// TIA Portal V17 export
// export: Created 2024-06-14T09:52:58.9808405Z, ExportSetting WithDefaults, DisplayName Totally Integrated Automation Portal, DisplayVersion V17, DisplayName TIA Portal Openness, DisplayVersion V17, DisplayName TIA Portal Version Control Interface, DisplayVersion V17, DisplayName Simotion SCOUT TIA, DisplayVersion 5.4.3.0, DisplayName SINAMICS Startdrive Advanced, DisplayVersion V17 SP1 Update 1, DisplayName SINAMICS Startdrive G110M, G120, G120C, G120D, G120P, G115D, DisplayVersion V17 SP1 Update 1, DisplayName SINAMICS Startdrive G130, G150, S120, S150, SINAMICS MV, S210, DisplayVersion V17 SP1 Update 1, DisplayName STEP 7 Professional, DisplayVersion V17, DisplayName STEP 7 Safety, DisplayVersion V17, DisplayName WinCC Professional, DisplayVersion V17
FUNCTION "STATION S1" : Void   // FC3, LAD
{ S7_Optimized_Access := 'TRUE' }
VERSION : 0.1
// stored: AutoNumber true, IsIECCheckEnabled false, SetENOAutomatically false, UDAEnableTagReadback false
   VAR_INPUT
      CYLINDER_POS_IN : Bool;
      INxcommercial_Cy : Bool;
      "CYLINDER EXIT" : Bool;
      sensor_line_1 : Bool;
      sensor_line_2 : Bool;
   END_VAR
   VAR_OUTPUT
      OUTxCylinder_Count : Bool;
      STOPPRER : Bool;
      Tare_Weight_Error : Bool;
      Enter_Tare_weight : Bool;
      Cylinder_type_error : Bool;
      data_count : Int;
   END_VAR
   VAR_IN_OUT
      S9_Array_copy : Int;
   END_VAR
   VAR_TEMP
      TRUCK : String;
      Start : Bool;
      copied_item : Int;
      Ret_val_1 : Int;
      Out_RD : DTL;
      Difference_Domestic_Cy : Real;
      Difference_commercial_Cy : Real;
      set_bit : Bool;
      Full_Wieght_Difference : Real;
      idx1 : Int;
      idx2 : Int;
      idx3 : Int;
      idx4 : Int;
      idx5 : Int;
      idx6 : Int;
      idx7 : Int;
      Gross_Weight : Real;
      "cylinder ok" : Bool;
      ptrig : Bool;
      ptrig_1 : Bool;
      ptrig_2 : Bool;
      TEMP : Int;
      pass : Bool;
      FILL_DB : Bool;
      TEMP_1 : Int;
      TEMP_2 : Int;
      TEMP_3 : Int;
      TEMP_4 : Int;
      TEMP_5 : Int;
      TEMP_6 : Int;
      TEMP_7 : Int;
      TEMP_8 : Int;
      TEMP_9 : Int;
      TEMP_10 : Int;
      TEMP_11 : Int;
      TEMP_12 : Int;
      TEMP_13 : Int;
      TEMP_14 : Int;
   END_VAR
   VAR_TEMP   // added for the SCL form of the ladder/FBD networks
      _w1 : Bool;
      _w2 : Bool;
      _w3 : Bool;
      _w4 : Bool;
      _w5 : Bool;
      _w6 : Bool;
      _w7 : Bool;
      _w8 : Bool;
      _w9 : Bool;
   END_VAR
BEGIN

REGION Network 1: Cylinder_Count
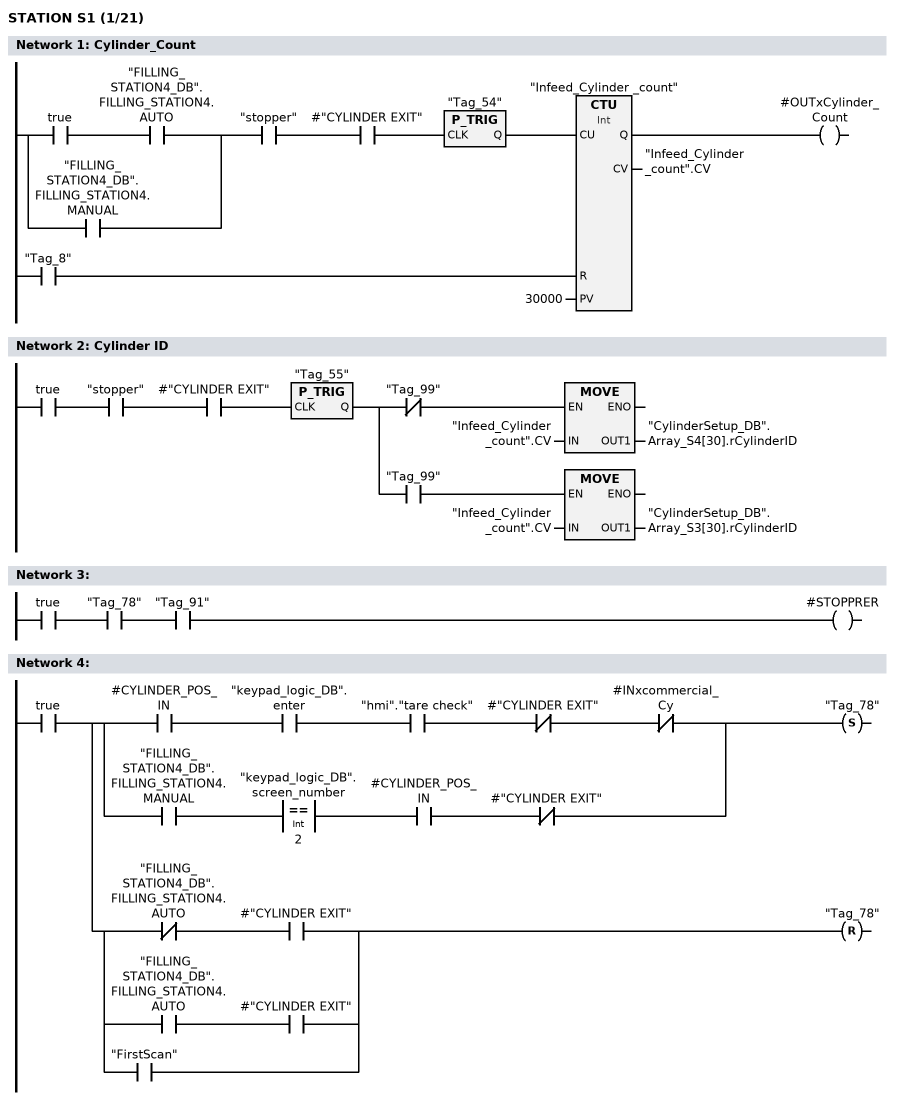
   RUNG wire#powerrail
      Contact( true )
      Contact( "FILLING_STATION4_DB".FILLING_STATION4.AUTO )
      wire#w1
      Contact( "stopper" )
      Contact( #"CYLINDER EXIT" )
      P_Trig( "Tag_54" )
      { S7_Templates := "value_type := Int" } "Infeed_Cylinder _count".CTU(r := wire#w2, pv := 30000, cv => "Infeed_Cylinder _count".CV)
      Coil( #OUTxCylinder_Count )
   END_RUNG
   RUNG wire#powerrail
      Contact( "FILLING_STATION4_DB".FILLING_STATION4.MANUAL )
   END_RUNG wire#w1
   RUNG wire#powerrail
      Contact( "Tag_8" )
   END_RUNG wire#w2
   // the same network as SCL:
   #_w1 := ((true AND "FILLING_STATION4_DB".FILLING_STATION4.AUTO) OR "FILLING_STATION4_DB".FILLING_STATION4.MANUAL) AND "stopper" AND #"CYLINDER EXIT";
   #_w2 := #_w1 AND NOT "Tag_54";   // rising edge
   "Tag_54" := #_w1;
   "Infeed_Cylinder _count".CTU(CU := #_w2, R := "Tag_8", PV := 30000, CV => "Infeed_Cylinder _count".CV);
   #OUTxCylinder_Count := "Infeed_Cylinder _count".Q;
END_REGION

REGION Network 2: Cylinder ID
   RUNG wire#powerrail
      Contact( true )
      Contact( "stopper" )
      Contact( #"CYLINDER EXIT" )
      P_Trig( "Tag_55" )
      wire#w1
      I_Contact( "Tag_99" )
      Move(in := "Infeed_Cylinder _count".CV, out1 => "CylinderSetup_DB".Array_S4[30].rCylinderID)
   END_RUNG
   RUNG wire#w1
      Contact( "Tag_99" )
      Move(in := "Infeed_Cylinder _count".CV, out1 => "CylinderSetup_DB".Array_S3[30].rCylinderID)
   END_RUNG
   // the same network as SCL:
   #_w1 := true AND "stopper" AND #"CYLINDER EXIT";
   #_w2 := #_w1 AND NOT "Tag_55";   // rising edge
   "Tag_55" := #_w1;
   IF #_w2 AND NOT "Tag_99" THEN
       "CylinderSetup_DB".Array_S4[30].rCylinderID := "Infeed_Cylinder _count".CV;
   END_IF;
   IF #_w2 AND "Tag_99" THEN
       "CylinderSetup_DB".Array_S3[30].rCylinderID := "Infeed_Cylinder _count".CV;
   END_IF;
END_REGION

REGION Network 3
   RUNG wire#powerrail
      Contact( true )
      Contact( "Tag_78" )
      Contact( "Tag_91" )
      Coil( #STOPPRER )
   END_RUNG
   // the same network as SCL:
   #STOPPRER := true AND "Tag_78" AND "Tag_91";
END_REGION

REGION Network 4
   RUNG wire#powerrail
      Contact( true )
      wire#w1
      Contact( #CYLINDER_POS_IN )
      Contact( "keypad_logic_DB".enter )
      Contact( "hmi"."tare check" )
      I_Contact( #"CYLINDER EXIT" )
      I_Contact( #INxcommercial_Cy )
      wire#w2
      S_Coil( "Tag_78" )
   END_RUNG
   RUNG wire#w1
      Contact( "FILLING_STATION4_DB".FILLING_STATION4.MANUAL )
      { S7_Templates := "SrcType := Int" } EQ_Contact(in1 := "keypad_logic_DB".screen_number, in2 := 2)
      Contact( #CYLINDER_POS_IN )
      I_Contact( #"CYLINDER EXIT" )
   END_RUNG wire#w2
   RUNG wire#w1
      I_Contact( "FILLING_STATION4_DB".FILLING_STATION4.AUTO )
      Contact( #"CYLINDER EXIT" )
      wire#w3
      R_Coil( "Tag_78" )
   END_RUNG
   RUNG wire#w1
      Contact( "FILLING_STATION4_DB".FILLING_STATION4.AUTO )
      Contact( #"CYLINDER EXIT" )
   END_RUNG wire#w3
   RUNG wire#w1
      Contact( "FirstScan" )
   END_RUNG wire#w3
   // the same network as SCL:
   IF true AND ((#CYLINDER_POS_IN AND "keypad_logic_DB".enter AND "hmi"."tare check" AND NOT #"CYLINDER EXIT" AND NOT #INxcommercial_Cy) OR ("FILLING_STATION4_DB".FILLING_STATION4.MANUAL AND ("keypad_logic_DB".screen_number = 2) AND #CYLINDER_POS_IN AND NOT #"CYLINDER EXIT")) THEN
       "Tag_78" := TRUE;
   END_IF;
   IF true AND ((NOT "FILLING_STATION4_DB".FILLING_STATION4.AUTO AND #"CYLINDER EXIT") OR ("FILLING_STATION4_DB".FILLING_STATION4.AUTO AND #"CYLINDER EXIT") OR "FirstScan") THEN
       "Tag_78" := FALSE;
   END_IF;
END_REGION

REGION Network 5: Domestic_Cylinder_Details
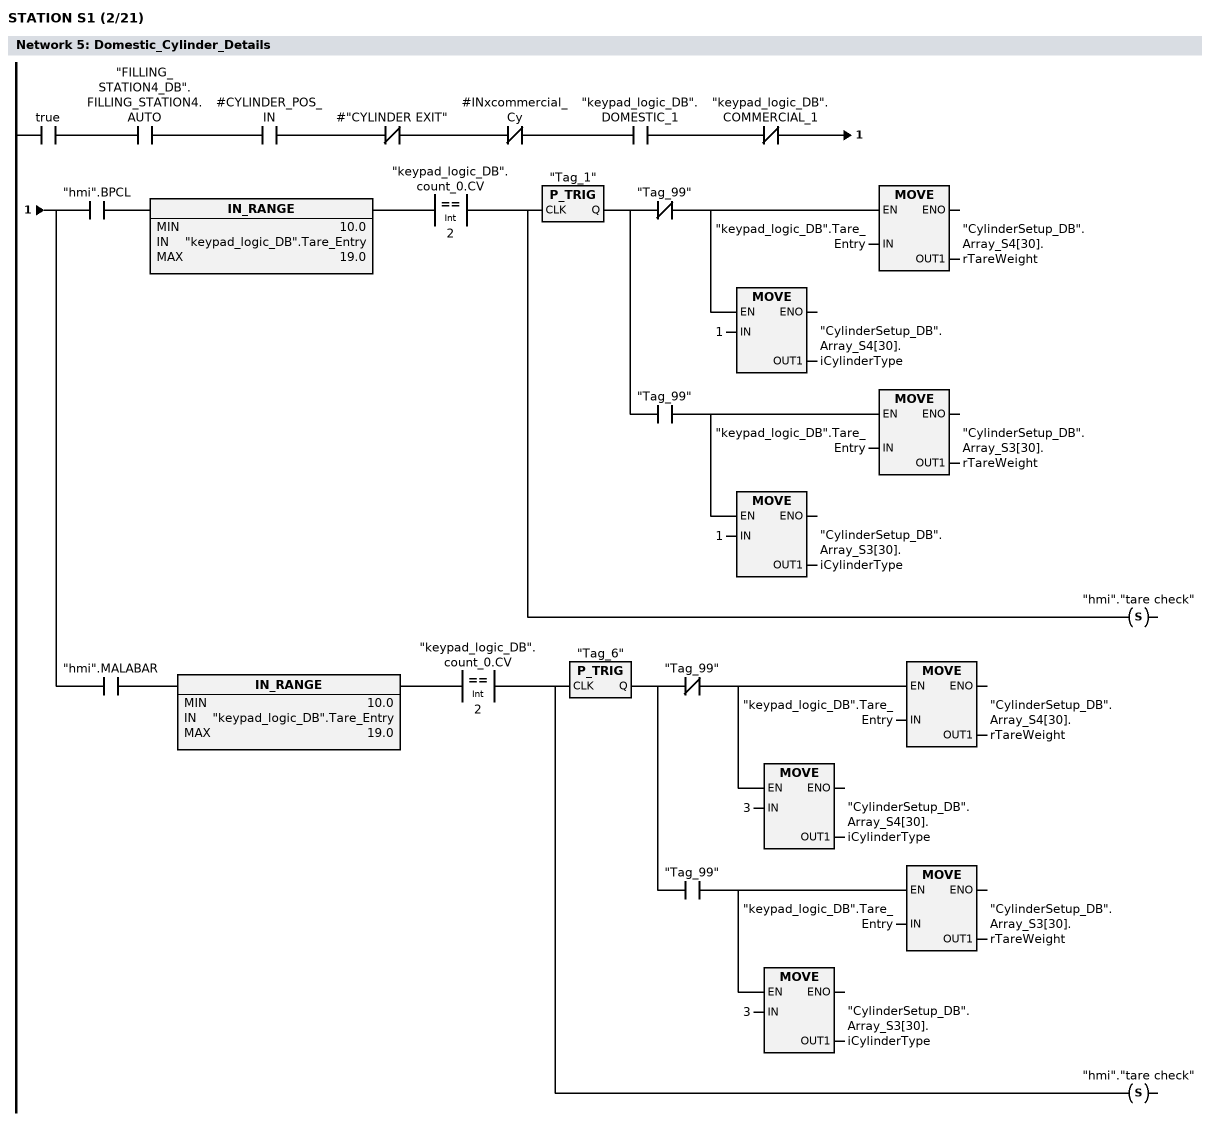
   RUNG wire#powerrail
      Contact( true )
      Contact( "FILLING_STATION4_DB".FILLING_STATION4.AUTO )
      Contact( #CYLINDER_POS_IN )
      I_Contact( #"CYLINDER EXIT" )
      I_Contact( #INxcommercial_Cy )
      Contact( "keypad_logic_DB".DOMESTIC_1 )
      I_Contact( "keypad_logic_DB".COMMERCIAL_1 )
      wire#w1
      Contact( "hmi".BPCL )
      { S7_Templates := "SrcType := Real" } InRange(min := 10.0, in := "keypad_logic_DB".Tare_Entry, max := 19.0)
      { S7_Templates := "SrcType := Int" } EQ_Contact(in1 := "keypad_logic_DB".count_0.CV, in2 := 2)
      wire#w2
      P_Trig( "Tag_1" )
      wire#w3
      I_Contact( "Tag_99" )
      wire#w4
      Move(in := "keypad_logic_DB".Tare_Entry, out1 => "CylinderSetup_DB".Array_S4[30].rTareWeight)
   END_RUNG
   RUNG wire#w4
      Move(in := 1, out1 => "CylinderSetup_DB".Array_S4[30].iCylinderType)
   END_RUNG
   RUNG wire#w3
      Contact( "Tag_99" )
      wire#w5
      Move(in := "keypad_logic_DB".Tare_Entry, out1 => "CylinderSetup_DB".Array_S3[30].rTareWeight)
   END_RUNG
   RUNG wire#w5
      Move(in := 1, out1 => "CylinderSetup_DB".Array_S3[30].iCylinderType)
   END_RUNG
   RUNG wire#w2
      S_Coil( "hmi"."tare check" )
   END_RUNG
   RUNG wire#w1
      Contact( "hmi".MALABAR )
      { S7_Templates := "SrcType := Real" } InRange(min := 10.0, in := "keypad_logic_DB".Tare_Entry, max := 19.0)
      { S7_Templates := "SrcType := Int" } EQ_Contact(in1 := "keypad_logic_DB".count_0.CV, in2 := 2)
      wire#w6
      P_Trig( "Tag_6" )
      wire#w7
      I_Contact( "Tag_99" )
      wire#w8
      Move(in := "keypad_logic_DB".Tare_Entry, out1 => "CylinderSetup_DB".Array_S4[30].rTareWeight)
   END_RUNG
   RUNG wire#w8
      Move(in := 3, out1 => "CylinderSetup_DB".Array_S4[30].iCylinderType)
   END_RUNG
   RUNG wire#w7
      Contact( "Tag_99" )
      wire#w9
      Move(in := "keypad_logic_DB".Tare_Entry, out1 => "CylinderSetup_DB".Array_S3[30].rTareWeight)
   END_RUNG
   RUNG wire#w9
      Move(in := 3, out1 => "CylinderSetup_DB".Array_S3[30].iCylinderType)
   END_RUNG
   RUNG wire#w6
      S_Coil( "hmi"."tare check" )
   END_RUNG
   // the same network as SCL:
   #_w1 := true AND "FILLING_STATION4_DB".FILLING_STATION4.AUTO AND #CYLINDER_POS_IN AND NOT #"CYLINDER EXIT" AND NOT #INxcommercial_Cy AND "keypad_logic_DB".DOMESTIC_1 AND NOT "keypad_logic_DB".COMMERCIAL_1;
   #_w2 := #_w1 AND "hmi".BPCL AND (10.0 <= "keypad_logic_DB".Tare_Entry) AND ("keypad_logic_DB".Tare_Entry <= 19.0) AND ("keypad_logic_DB".count_0.CV = 2);
   #_w3 := #_w2 AND NOT "Tag_1";   // rising edge
   "Tag_1" := #_w2;
   IF #_w3 AND NOT "Tag_99" THEN
       "CylinderSetup_DB".Array_S4[30].rTareWeight := "keypad_logic_DB".Tare_Entry;
       "CylinderSetup_DB".Array_S4[30].iCylinderType := 1;
   END_IF;
   IF #_w3 AND "Tag_99" THEN
       "CylinderSetup_DB".Array_S3[30].rTareWeight := "keypad_logic_DB".Tare_Entry;
       "CylinderSetup_DB".Array_S3[30].iCylinderType := 1;
   END_IF;
   IF #_w2 THEN "hmi"."tare check" := TRUE; END_IF;
   #_w4 := #_w1 AND "hmi".MALABAR AND (10.0 <= "keypad_logic_DB".Tare_Entry) AND ("keypad_logic_DB".Tare_Entry <= 19.0) AND ("keypad_logic_DB".count_0.CV = 2);
   #_w5 := #_w4 AND NOT "Tag_6";   // rising edge
   "Tag_6" := #_w4;
   IF #_w5 AND NOT "Tag_99" THEN
       "CylinderSetup_DB".Array_S4[30].rTareWeight := "keypad_logic_DB".Tare_Entry;
       "CylinderSetup_DB".Array_S4[30].iCylinderType := 3;
   END_IF;
   IF #_w5 AND "Tag_99" THEN
       "CylinderSetup_DB".Array_S3[30].rTareWeight := "keypad_logic_DB".Tare_Entry;
       "CylinderSetup_DB".Array_S3[30].iCylinderType := 3;
   END_IF;
   IF #_w4 THEN "hmi"."tare check" := TRUE; END_IF;
END_REGION

REGION Network 6: DOMESTIC_ALARM
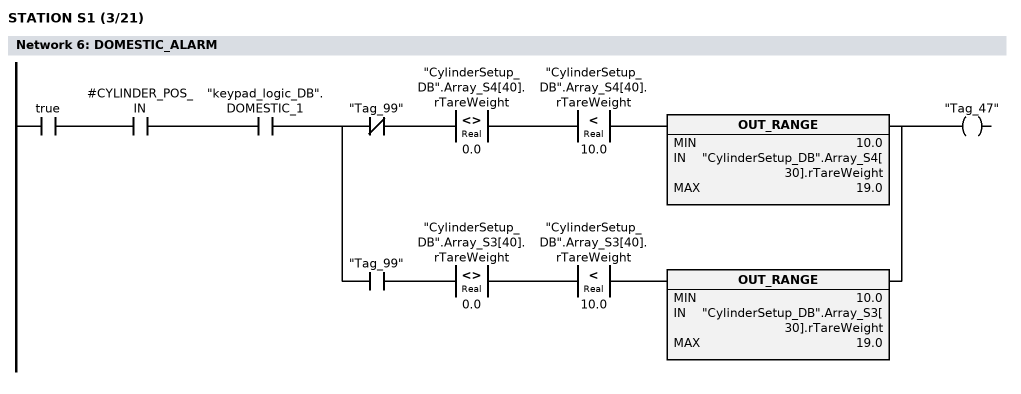
   "Tag_47" := true AND #CYLINDER_POS_IN AND "keypad_logic_DB".DOMESTIC_1 AND ((NOT "Tag_99" AND ("CylinderSetup_DB".Array_S4[40].rTareWeight <> 0.0) AND ("CylinderSetup_DB".Array_S4[40].rTareWeight < 10.0) AND (("CylinderSetup_DB".Array_S4[30].rTareWeight < 10.0) OR ("CylinderSetup_DB".Array_S4[30].rTareWeight > 19.0))) OR ("Tag_99" AND ("CylinderSetup_DB".Array_S3[40].rTareWeight <> 0.0) AND ("CylinderSetup_DB".Array_S3[40].rTareWeight < 10.0) AND (("CylinderSetup_DB".Array_S3[30].rTareWeight < 10.0) OR ("CylinderSetup_DB".Array_S3[30].rTareWeight > 19.0))));
END_REGION

REGION Network 7: Commercial_Cylinder_Details
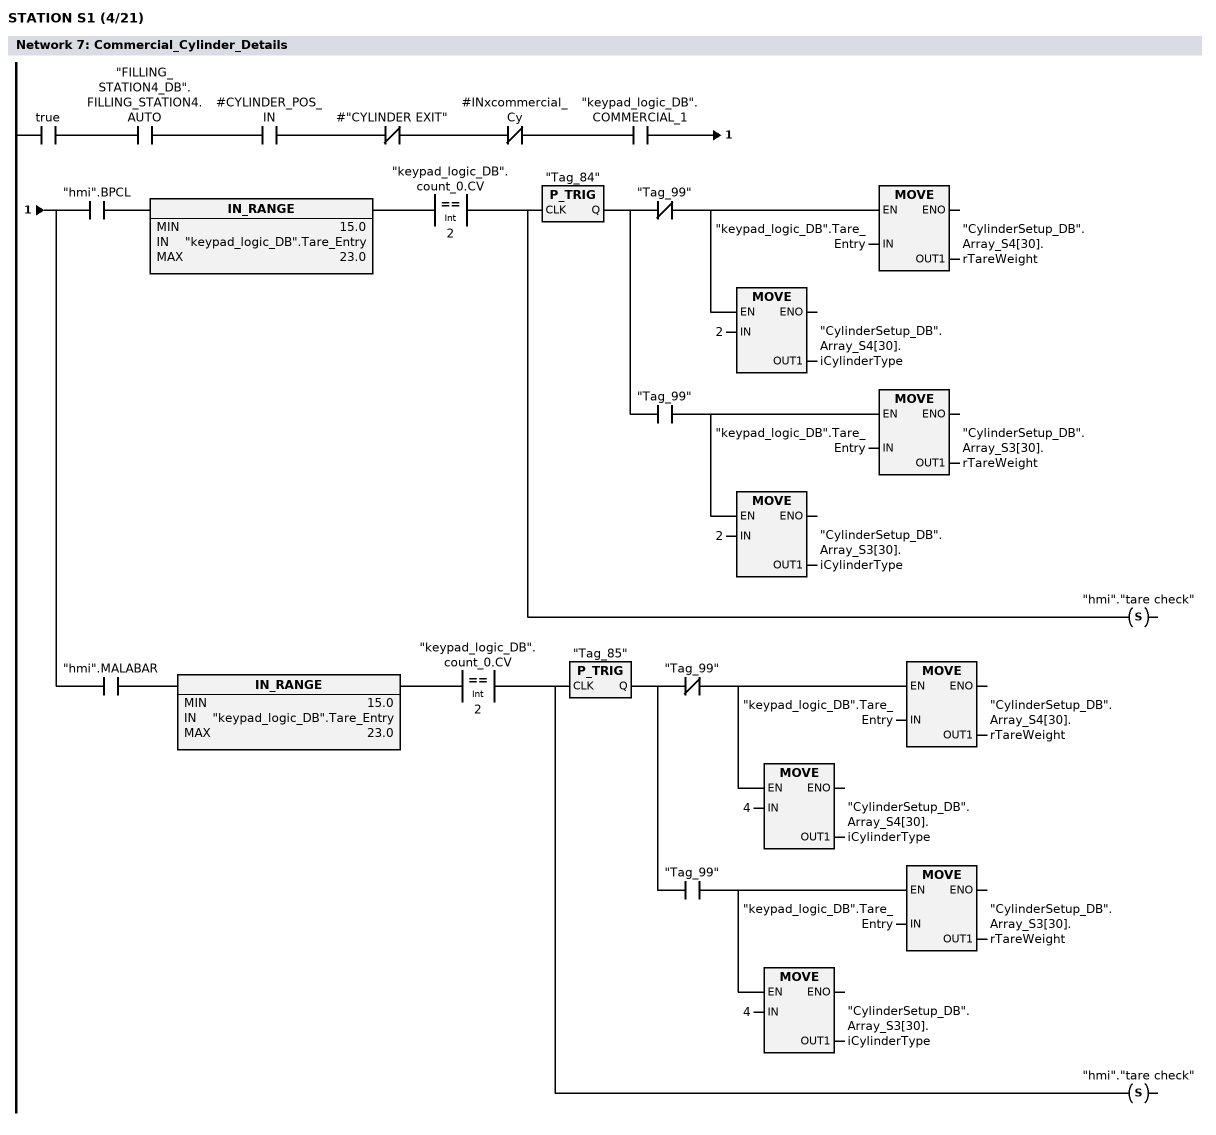
   RUNG wire#powerrail
      Contact( true )
      Contact( "FILLING_STATION4_DB".FILLING_STATION4.AUTO )
      Contact( #CYLINDER_POS_IN )
      I_Contact( #"CYLINDER EXIT" )
      I_Contact( #INxcommercial_Cy )
      Contact( "keypad_logic_DB".COMMERCIAL_1 )
      wire#w1
      Contact( "hmi".BPCL )
      { S7_Templates := "SrcType := Real" } InRange(min := 15.0, in := "keypad_logic_DB".Tare_Entry, max := 23.0)
      { S7_Templates := "SrcType := Int" } EQ_Contact(in1 := "keypad_logic_DB".count_0.CV, in2 := 2)
      wire#w2
      P_Trig( "Tag_84" )
      wire#w3
      I_Contact( "Tag_99" )
      wire#w4
      Move(in := "keypad_logic_DB".Tare_Entry, out1 => "CylinderSetup_DB".Array_S4[30].rTareWeight)
   END_RUNG
   RUNG wire#w4
      Move(in := 2, out1 => "CylinderSetup_DB".Array_S4[30].iCylinderType)
   END_RUNG
   RUNG wire#w3
      Contact( "Tag_99" )
      wire#w5
      Move(in := "keypad_logic_DB".Tare_Entry, out1 => "CylinderSetup_DB".Array_S3[30].rTareWeight)
   END_RUNG
   RUNG wire#w5
      Move(in := 2, out1 => "CylinderSetup_DB".Array_S3[30].iCylinderType)
   END_RUNG
   RUNG wire#w2
      S_Coil( "hmi"."tare check" )
   END_RUNG
   RUNG wire#w1
      Contact( "hmi".MALABAR )
      { S7_Templates := "SrcType := Real" } InRange(min := 15.0, in := "keypad_logic_DB".Tare_Entry, max := 23.0)
      { S7_Templates := "SrcType := Int" } EQ_Contact(in1 := "keypad_logic_DB".count_0.CV, in2 := 2)
      wire#w6
      P_Trig( "Tag_85" )
      wire#w7
      I_Contact( "Tag_99" )
      wire#w8
      Move(in := "keypad_logic_DB".Tare_Entry, out1 => "CylinderSetup_DB".Array_S4[30].rTareWeight)
   END_RUNG
   RUNG wire#w8
      Move(in := 4, out1 => "CylinderSetup_DB".Array_S4[30].iCylinderType)
   END_RUNG
   RUNG wire#w7
      Contact( "Tag_99" )
      wire#w9
      Move(in := "keypad_logic_DB".Tare_Entry, out1 => "CylinderSetup_DB".Array_S3[30].rTareWeight)
   END_RUNG
   RUNG wire#w9
      Move(in := 4, out1 => "CylinderSetup_DB".Array_S3[30].iCylinderType)
   END_RUNG
   RUNG wire#w6
      S_Coil( "hmi"."tare check" )
   END_RUNG
   // the same network as SCL:
   #_w1 := true AND "FILLING_STATION4_DB".FILLING_STATION4.AUTO AND #CYLINDER_POS_IN AND NOT #"CYLINDER EXIT" AND NOT #INxcommercial_Cy AND "keypad_logic_DB".COMMERCIAL_1;
   #_w2 := #_w1 AND "hmi".BPCL AND (15.0 <= "keypad_logic_DB".Tare_Entry) AND ("keypad_logic_DB".Tare_Entry <= 23.0) AND ("keypad_logic_DB".count_0.CV = 2);
   #_w3 := #_w2 AND NOT "Tag_84";   // rising edge
   "Tag_84" := #_w2;
   IF #_w3 AND NOT "Tag_99" THEN
       "CylinderSetup_DB".Array_S4[30].rTareWeight := "keypad_logic_DB".Tare_Entry;
       "CylinderSetup_DB".Array_S4[30].iCylinderType := 2;
   END_IF;
   IF #_w3 AND "Tag_99" THEN
       "CylinderSetup_DB".Array_S3[30].rTareWeight := "keypad_logic_DB".Tare_Entry;
       "CylinderSetup_DB".Array_S3[30].iCylinderType := 2;
   END_IF;
   IF #_w2 THEN "hmi"."tare check" := TRUE; END_IF;
   #_w4 := #_w1 AND "hmi".MALABAR AND (15.0 <= "keypad_logic_DB".Tare_Entry) AND ("keypad_logic_DB".Tare_Entry <= 23.0) AND ("keypad_logic_DB".count_0.CV = 2);
   #_w5 := #_w4 AND NOT "Tag_85";   // rising edge
   "Tag_85" := #_w4;
   IF #_w5 AND NOT "Tag_99" THEN
       "CylinderSetup_DB".Array_S4[30].rTareWeight := "keypad_logic_DB".Tare_Entry;
       "CylinderSetup_DB".Array_S4[30].iCylinderType := 4;
   END_IF;
   IF #_w5 AND "Tag_99" THEN
       "CylinderSetup_DB".Array_S3[30].rTareWeight := "keypad_logic_DB".Tare_Entry;
       "CylinderSetup_DB".Array_S3[30].iCylinderType := 4;
   END_IF;
   IF #_w4 THEN "hmi"."tare check" := TRUE; END_IF;
END_REGION

REGION Network 8: COMMERCIAL_ALARM
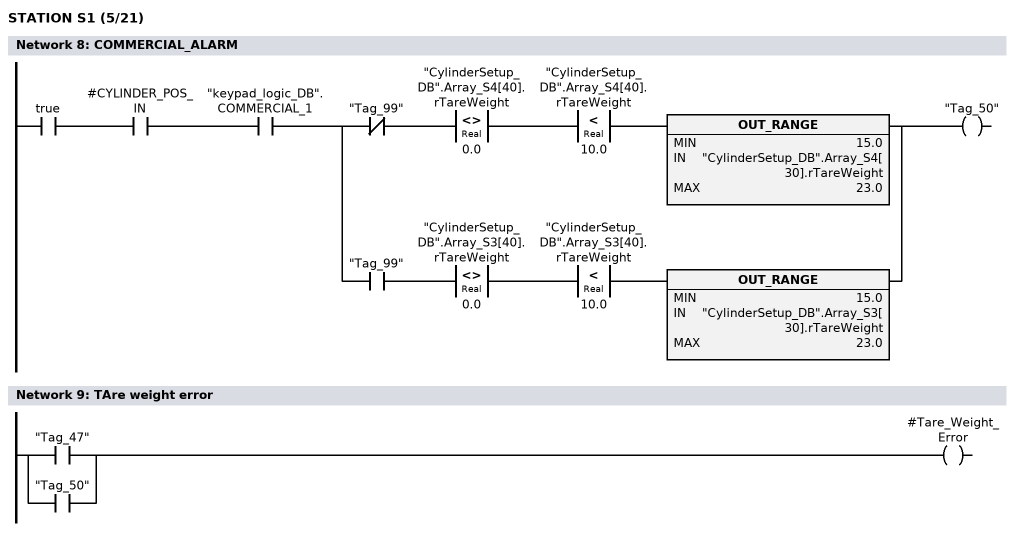
   "Tag_50" := true AND #CYLINDER_POS_IN AND "keypad_logic_DB".COMMERCIAL_1 AND ((NOT "Tag_99" AND ("CylinderSetup_DB".Array_S4[40].rTareWeight <> 0.0) AND ("CylinderSetup_DB".Array_S4[40].rTareWeight < 10.0) AND (("CylinderSetup_DB".Array_S4[30].rTareWeight < 15.0) OR ("CylinderSetup_DB".Array_S4[30].rTareWeight > 23.0))) OR ("Tag_99" AND ("CylinderSetup_DB".Array_S3[40].rTareWeight <> 0.0) AND ("CylinderSetup_DB".Array_S3[40].rTareWeight < 10.0) AND (("CylinderSetup_DB".Array_S3[30].rTareWeight < 15.0) OR ("CylinderSetup_DB".Array_S3[30].rTareWeight > 23.0))));
END_REGION

REGION Network 9: TAre weight error
   RUNG wire#powerrail
      Contact( "Tag_47" )
      wire#w1
      Coil( #Tare_Weight_Error )
   END_RUNG
   RUNG wire#powerrail
      Contact( "Tag_50" )
   END_RUNG wire#w1
   // the same network as SCL:
   #Tare_Weight_Error := "Tag_47" OR "Tag_50";
END_REGION

REGION Network 10: S4_Array Move
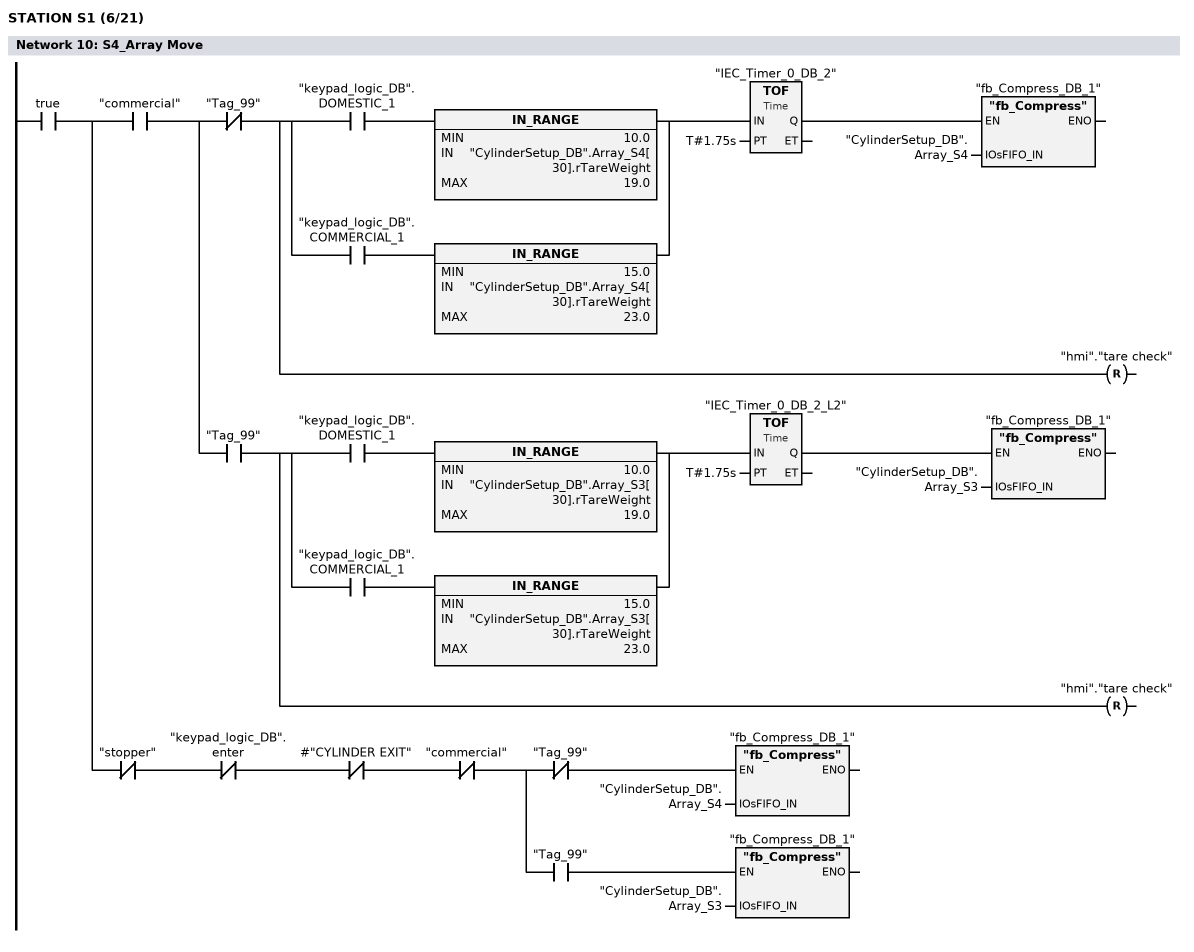
   RUNG wire#powerrail
      Contact( true )
      wire#w1
      Contact( "commercial" )
      wire#w2
      I_Contact( "Tag_99" )
      wire#w3
      Contact( "keypad_logic_DB".DOMESTIC_1 )
      { S7_Templates := "SrcType := Real" } InRange(min := 10.0, in := "CylinderSetup_DB".Array_S4[30].rTareWeight, max := 19.0)
      wire#w4
      { S7_Templates := "time_type := Time" } "IEC_Timer_0_DB_2".TOF(pt := T#1.75s, et =>)
      "fb_Compress_DB_1"(IOsFIFO_IN := "CylinderSetup_DB".Array_S4)
   END_RUNG
   RUNG wire#w3
      Contact( "keypad_logic_DB".COMMERCIAL_1 )
      { S7_Templates := "SrcType := Real" } InRange(min := 15.0, in := "CylinderSetup_DB".Array_S4[30].rTareWeight, max := 23.0)
   END_RUNG wire#w4
   RUNG wire#w3
      R_Coil( "hmi"."tare check" )
   END_RUNG
   RUNG wire#w2
      Contact( "Tag_99" )
      wire#w5
      Contact( "keypad_logic_DB".DOMESTIC_1 )
      { S7_Templates := "SrcType := Real" } InRange(min := 10.0, in := "CylinderSetup_DB".Array_S3[30].rTareWeight, max := 19.0)
      wire#w6
      { S7_Templates := "time_type := Time" } "IEC_Timer_0_DB_2_L2".TOF(pt := T#1.75s, et =>)
      "fb_Compress_DB_1"(IOsFIFO_IN := "CylinderSetup_DB".Array_S3)
   END_RUNG
   RUNG wire#w5
      Contact( "keypad_logic_DB".COMMERCIAL_1 )
      { S7_Templates := "SrcType := Real" } InRange(min := 15.0, in := "CylinderSetup_DB".Array_S3[30].rTareWeight, max := 23.0)
   END_RUNG wire#w6
   RUNG wire#w5
      R_Coil( "hmi"."tare check" )
   END_RUNG
   RUNG wire#w1
      I_Contact( "stopper" )
      I_Contact( "keypad_logic_DB".enter )
      I_Contact( #"CYLINDER EXIT" )
      I_Contact( "commercial" )
      wire#w7
      I_Contact( "Tag_99" )
      "fb_Compress_DB_1"(IOsFIFO_IN := "CylinderSetup_DB".Array_S4)
   END_RUNG
   RUNG wire#w7
      Contact( "Tag_99" )
      "fb_Compress_DB_1"(IOsFIFO_IN := "CylinderSetup_DB".Array_S3)
   END_RUNG
   // the same network as SCL:
   #_w1 := true AND "commercial";
   #_w2 := #_w1 AND NOT "Tag_99";
   "IEC_Timer_0_DB_2".TOF(IN := #_w2 AND (("keypad_logic_DB".DOMESTIC_1 AND (10.0 <= "CylinderSetup_DB".Array_S4[30].rTareWeight) AND ("CylinderSetup_DB".Array_S4[30].rTareWeight <= 19.0)) OR ("keypad_logic_DB".COMMERCIAL_1 AND (15.0 <= "CylinderSetup_DB".Array_S4[30].rTareWeight) AND ("CylinderSetup_DB".Array_S4[30].rTareWeight <= 23.0))),
                          PT := T#1.75s);
   IF "IEC_Timer_0_DB_2".Q THEN
       "fb_Compress_DB_1"(IOsFIFO_IN := "CylinderSetup_DB".Array_S4);   // "fb_Compress"
   END_IF;
   IF #_w2 THEN "hmi"."tare check" := FALSE; END_IF;
   #_w3 := #_w1 AND "Tag_99";
   "IEC_Timer_0_DB_2_L2".TOF(IN := #_w3 AND (("keypad_logic_DB".DOMESTIC_1 AND (10.0 <= "CylinderSetup_DB".Array_S3[30].rTareWeight) AND ("CylinderSetup_DB".Array_S3[30].rTareWeight <= 19.0)) OR ("keypad_logic_DB".COMMERCIAL_1 AND (15.0 <= "CylinderSetup_DB".Array_S3[30].rTareWeight) AND ("CylinderSetup_DB".Array_S3[30].rTareWeight <= 23.0))),
                           PT := T#1.75s);
   IF "IEC_Timer_0_DB_2_L2".Q THEN
       "fb_Compress_DB_1"(IOsFIFO_IN := "CylinderSetup_DB".Array_S3);   // "fb_Compress"
   END_IF;
   IF #_w3 THEN "hmi"."tare check" := FALSE; END_IF;
   #_w4 := true AND NOT "stopper" AND NOT "keypad_logic_DB".enter AND NOT #"CYLINDER EXIT" AND NOT "commercial";
   IF #_w4 AND NOT "Tag_99" THEN
       "fb_Compress_DB_1"(IOsFIFO_IN := "CylinderSetup_DB".Array_S4);   // "fb_Compress"
   END_IF;
   IF #_w4 AND "Tag_99" THEN
       "fb_Compress_DB_1"(IOsFIFO_IN := "CylinderSetup_DB".Array_S3);   // "fb_Compress"
   END_IF;
END_REGION

REGION Network 11: Station1_Rejection NOT USE
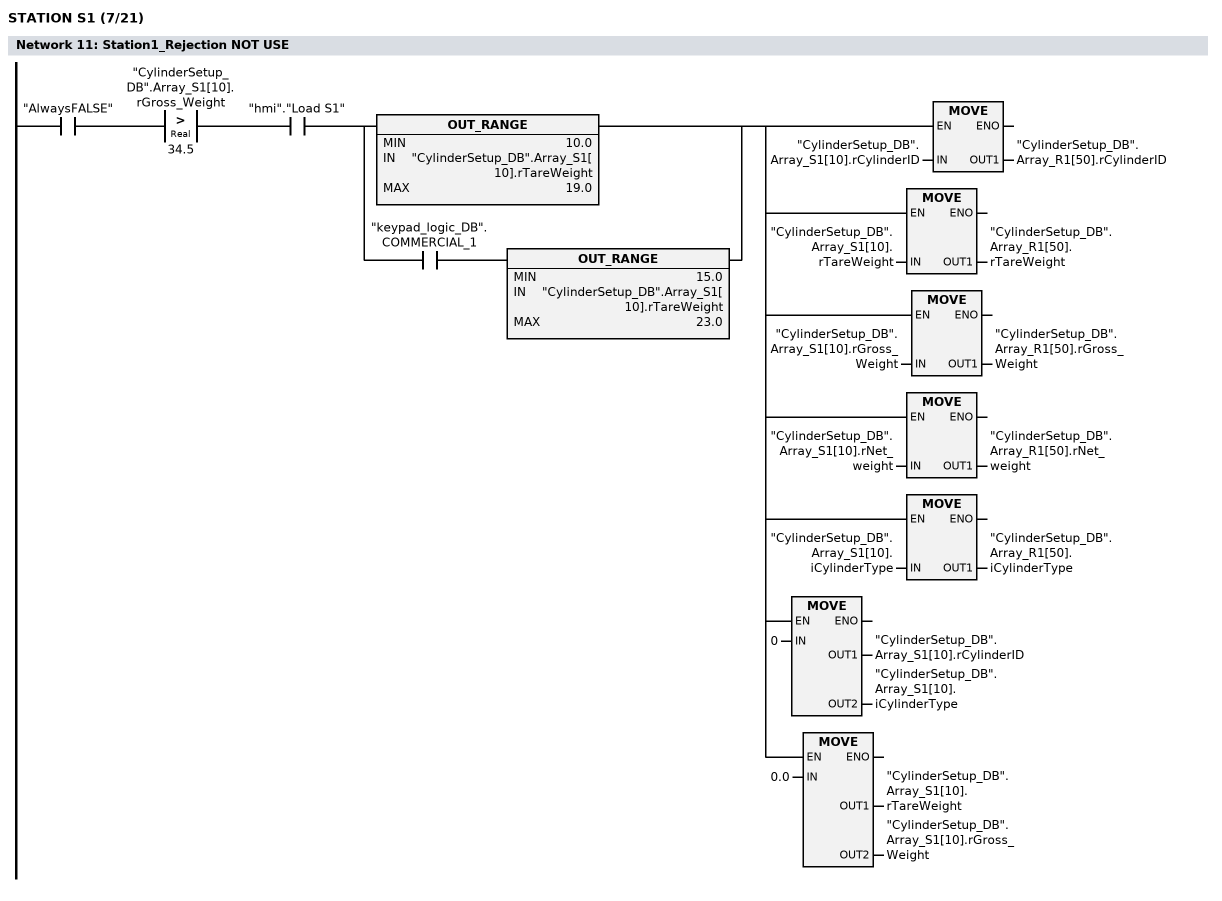
   IF "AlwaysFALSE" AND ("CylinderSetup_DB".Array_S1[10].rGross_Weight > 34.5) AND "hmi"."Load S1" AND (("CylinderSetup_DB".Array_S1[10].rTareWeight < 10.0) OR ("CylinderSetup_DB".Array_S1[10].rTareWeight > 19.0) OR ("keypad_logic_DB".COMMERCIAL_1 AND (("CylinderSetup_DB".Array_S1[10].rTareWeight < 15.0) OR ("CylinderSetup_DB".Array_S1[10].rTareWeight > 23.0)))) THEN
       "CylinderSetup_DB".Array_R1[50].rCylinderID := "CylinderSetup_DB".Array_S1[10].rCylinderID;
       "CylinderSetup_DB".Array_R1[50].rTareWeight := "CylinderSetup_DB".Array_S1[10].rTareWeight;
       "CylinderSetup_DB".Array_R1[50].rGross_Weight := "CylinderSetup_DB".Array_S1[10].rGross_Weight;
       "CylinderSetup_DB".Array_R1[50].rNet_weight := "CylinderSetup_DB".Array_S1[10].rNet_weight;
       "CylinderSetup_DB".Array_R1[50].iCylinderType := "CylinderSetup_DB".Array_S1[10].iCylinderType;
   END_IF;
   #_w1 := "AlwaysFALSE" AND ("CylinderSetup_DB".Array_S1[10].rGross_Weight > 34.5) AND "hmi"."Load S1" AND (("CylinderSetup_DB".Array_S1[10].rTareWeight < 10.0) OR ("CylinderSetup_DB".Array_S1[10].rTareWeight > 19.0) OR ("keypad_logic_DB".COMMERCIAL_1 AND (("CylinderSetup_DB".Array_S1[10].rTareWeight < 15.0) OR ("CylinderSetup_DB".Array_S1[10].rTareWeight > 23.0))));
   IF #_w1 THEN
       "CylinderSetup_DB".Array_S1[10].rCylinderID := 0;
       "CylinderSetup_DB".Array_S1[10].iCylinderType := 0;
       "CylinderSetup_DB".Array_S1[10].rTareWeight := 0.0;
       "CylinderSetup_DB".Array_S1[10].rGross_Weight := 0.0;
   END_IF;
END_REGION

REGION Network 12: data move
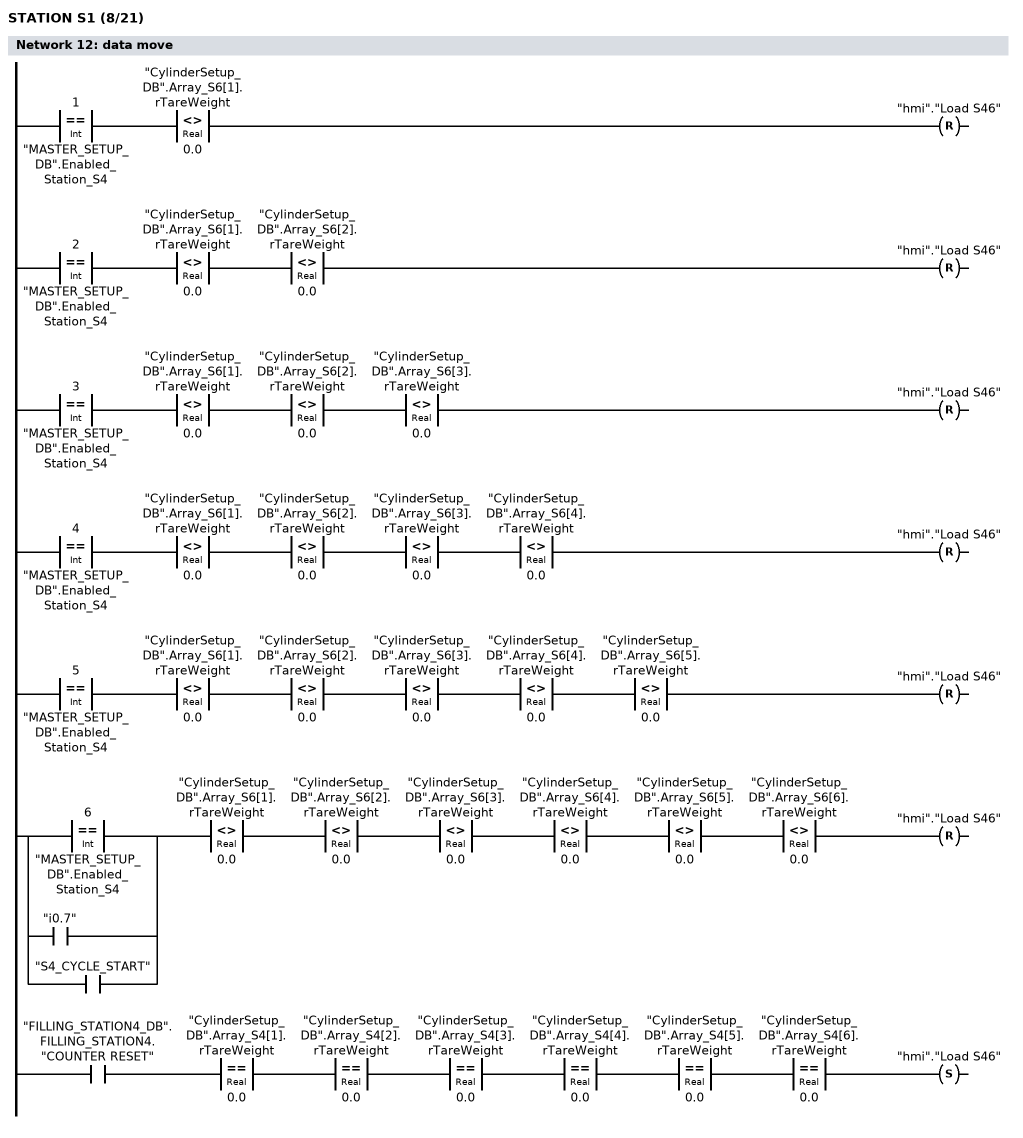
   RUNG wire#powerrail
      { S7_Templates := "SrcType := Int" } EQ_Contact(in1 := 1, in2 := "MASTER_SETUP_DB".Enabled_Station_S4)
      { S7_Templates := "SrcType := Real" } NE_Contact(in1 := "CylinderSetup_DB".Array_S6[1].rTareWeight, in2 := 0.0)
      R_Coil( "hmi"."Load S46" )
   END_RUNG
   RUNG wire#powerrail
      { S7_Templates := "SrcType := Int" } EQ_Contact(in1 := 2, in2 := "MASTER_SETUP_DB".Enabled_Station_S4)
      { S7_Templates := "SrcType := Real" } NE_Contact(in1 := "CylinderSetup_DB".Array_S6[1].rTareWeight, in2 := 0.0)
      { S7_Templates := "SrcType := Real" } NE_Contact(in1 := "CylinderSetup_DB".Array_S6[2].rTareWeight, in2 := 0.0)
      R_Coil( "hmi"."Load S46" )
   END_RUNG
   RUNG wire#powerrail
      { S7_Templates := "SrcType := Int" } EQ_Contact(in1 := 3, in2 := "MASTER_SETUP_DB".Enabled_Station_S4)
      { S7_Templates := "SrcType := Real" } NE_Contact(in1 := "CylinderSetup_DB".Array_S6[1].rTareWeight, in2 := 0.0)
      { S7_Templates := "SrcType := Real" } NE_Contact(in1 := "CylinderSetup_DB".Array_S6[2].rTareWeight, in2 := 0.0)
      { S7_Templates := "SrcType := Real" } NE_Contact(in1 := "CylinderSetup_DB".Array_S6[3].rTareWeight, in2 := 0.0)
      R_Coil( "hmi"."Load S46" )
   END_RUNG
   RUNG wire#powerrail
      { S7_Templates := "SrcType := Int" } EQ_Contact(in1 := 4, in2 := "MASTER_SETUP_DB".Enabled_Station_S4)
      { S7_Templates := "SrcType := Real" } NE_Contact(in1 := "CylinderSetup_DB".Array_S6[1].rTareWeight, in2 := 0.0)
      { S7_Templates := "SrcType := Real" } NE_Contact(in1 := "CylinderSetup_DB".Array_S6[2].rTareWeight, in2 := 0.0)
      { S7_Templates := "SrcType := Real" } NE_Contact(in1 := "CylinderSetup_DB".Array_S6[3].rTareWeight, in2 := 0.0)
      { S7_Templates := "SrcType := Real" } NE_Contact(in1 := "CylinderSetup_DB".Array_S6[4].rTareWeight, in2 := 0.0)
      R_Coil( "hmi"."Load S46" )
   END_RUNG
   RUNG wire#powerrail
      { S7_Templates := "SrcType := Int" } EQ_Contact(in1 := 5, in2 := "MASTER_SETUP_DB".Enabled_Station_S4)
      { S7_Templates := "SrcType := Real" } NE_Contact(in1 := "CylinderSetup_DB".Array_S6[1].rTareWeight, in2 := 0.0)
      { S7_Templates := "SrcType := Real" } NE_Contact(in1 := "CylinderSetup_DB".Array_S6[2].rTareWeight, in2 := 0.0)
      { S7_Templates := "SrcType := Real" } NE_Contact(in1 := "CylinderSetup_DB".Array_S6[3].rTareWeight, in2 := 0.0)
      { S7_Templates := "SrcType := Real" } NE_Contact(in1 := "CylinderSetup_DB".Array_S6[4].rTareWeight, in2 := 0.0)
      { S7_Templates := "SrcType := Real" } NE_Contact(in1 := "CylinderSetup_DB".Array_S6[5].rTareWeight, in2 := 0.0)
      R_Coil( "hmi"."Load S46" )
   END_RUNG
   RUNG wire#powerrail
      { S7_Templates := "SrcType := Int" } EQ_Contact(in1 := 6, in2 := "MASTER_SETUP_DB".Enabled_Station_S4)
      wire#w1
      { S7_Templates := "SrcType := Real" } NE_Contact(in1 := "CylinderSetup_DB".Array_S6[1].rTareWeight, in2 := 0.0)
      { S7_Templates := "SrcType := Real" } NE_Contact(in1 := "CylinderSetup_DB".Array_S6[2].rTareWeight, in2 := 0.0)
      { S7_Templates := "SrcType := Real" } NE_Contact(in1 := "CylinderSetup_DB".Array_S6[3].rTareWeight, in2 := 0.0)
      { S7_Templates := "SrcType := Real" } NE_Contact(in1 := "CylinderSetup_DB".Array_S6[4].rTareWeight, in2 := 0.0)
      { S7_Templates := "SrcType := Real" } NE_Contact(in1 := "CylinderSetup_DB".Array_S6[5].rTareWeight, in2 := 0.0)
      { S7_Templates := "SrcType := Real" } NE_Contact(in1 := "CylinderSetup_DB".Array_S6[6].rTareWeight, in2 := 0.0)
      R_Coil( "hmi"."Load S46" )
   END_RUNG
   RUNG wire#powerrail
      Contact( "i0.7" )
   END_RUNG wire#w1
   RUNG wire#powerrail
      Contact( "S4_CYCLE_START" )
   END_RUNG wire#w1
   RUNG wire#powerrail
      Contact( "FILLING_STATION4_DB".FILLING_STATION4."COUNTER RESET" )
      { S7_Templates := "SrcType := Real" } EQ_Contact(in1 := "CylinderSetup_DB".Array_S4[1].rTareWeight, in2 := 0.0)
      { S7_Templates := "SrcType := Real" } EQ_Contact(in1 := "CylinderSetup_DB".Array_S4[2].rTareWeight, in2 := 0.0)
      { S7_Templates := "SrcType := Real" } EQ_Contact(in1 := "CylinderSetup_DB".Array_S4[3].rTareWeight, in2 := 0.0)
      { S7_Templates := "SrcType := Real" } EQ_Contact(in1 := "CylinderSetup_DB".Array_S4[4].rTareWeight, in2 := 0.0)
      { S7_Templates := "SrcType := Real" } EQ_Contact(in1 := "CylinderSetup_DB".Array_S4[5].rTareWeight, in2 := 0.0)
      { S7_Templates := "SrcType := Real" } EQ_Contact(in1 := "CylinderSetup_DB".Array_S4[6].rTareWeight, in2 := 0.0)
      S_Coil( "hmi"."Load S46" )
   END_RUNG
   // the same network as SCL:
   IF (1 = "MASTER_SETUP_DB".Enabled_Station_S4) AND ("CylinderSetup_DB".Array_S6[1].rTareWeight <> 0.0) THEN
       "hmi"."Load S46" := FALSE;
   END_IF;
   IF (2 = "MASTER_SETUP_DB".Enabled_Station_S4) AND ("CylinderSetup_DB".Array_S6[1].rTareWeight <> 0.0) AND ("CylinderSetup_DB".Array_S6[2].rTareWeight <> 0.0) THEN
       "hmi"."Load S46" := FALSE;
   END_IF;
   IF (3 = "MASTER_SETUP_DB".Enabled_Station_S4) AND ("CylinderSetup_DB".Array_S6[1].rTareWeight <> 0.0) AND ("CylinderSetup_DB".Array_S6[2].rTareWeight <> 0.0) AND ("CylinderSetup_DB".Array_S6[3].rTareWeight <> 0.0) THEN
       "hmi"."Load S46" := FALSE;
   END_IF;
   IF (4 = "MASTER_SETUP_DB".Enabled_Station_S4) AND ("CylinderSetup_DB".Array_S6[1].rTareWeight <> 0.0) AND ("CylinderSetup_DB".Array_S6[2].rTareWeight <> 0.0) AND ("CylinderSetup_DB".Array_S6[3].rTareWeight <> 0.0) AND ("CylinderSetup_DB".Array_S6[4].rTareWeight <> 0.0) THEN
       "hmi"."Load S46" := FALSE;
   END_IF;
   IF (5 = "MASTER_SETUP_DB".Enabled_Station_S4) AND ("CylinderSetup_DB".Array_S6[1].rTareWeight <> 0.0) AND ("CylinderSetup_DB".Array_S6[2].rTareWeight <> 0.0) AND ("CylinderSetup_DB".Array_S6[3].rTareWeight <> 0.0) AND ("CylinderSetup_DB".Array_S6[4].rTareWeight <> 0.0) AND ("CylinderSetup_DB".Array_S6[5].rTareWeight <> 0.0) THEN
       "hmi"."Load S46" := FALSE;
   END_IF;
   IF ((6 = "MASTER_SETUP_DB".Enabled_Station_S4) OR "i0.7" OR "S4_CYCLE_START") AND ("CylinderSetup_DB".Array_S6[1].rTareWeight <> 0.0) AND ("CylinderSetup_DB".Array_S6[2].rTareWeight <> 0.0) AND ("CylinderSetup_DB".Array_S6[3].rTareWeight <> 0.0) AND ("CylinderSetup_DB".Array_S6[4].rTareWeight <> 0.0) AND ("CylinderSetup_DB".Array_S6[5].rTareWeight <> 0.0) AND ("CylinderSetup_DB".Array_S6[6].rTareWeight <> 0.0) THEN
       "hmi"."Load S46" := FALSE;
   END_IF;
   IF "FILLING_STATION4_DB".FILLING_STATION4."COUNTER RESET" AND ("CylinderSetup_DB".Array_S4[1].rTareWeight = 0.0) AND ("CylinderSetup_DB".Array_S4[2].rTareWeight = 0.0) AND ("CylinderSetup_DB".Array_S4[3].rTareWeight = 0.0) AND ("CylinderSetup_DB".Array_S4[4].rTareWeight = 0.0) AND ("CylinderSetup_DB".Array_S4[5].rTareWeight = 0.0) AND ("CylinderSetup_DB".Array_S4[6].rTareWeight = 0.0) THEN
       "hmi"."Load S46" := TRUE;
   END_IF;
END_REGION

REGION Network 13: S6_TO_S8 SAME L1 exit
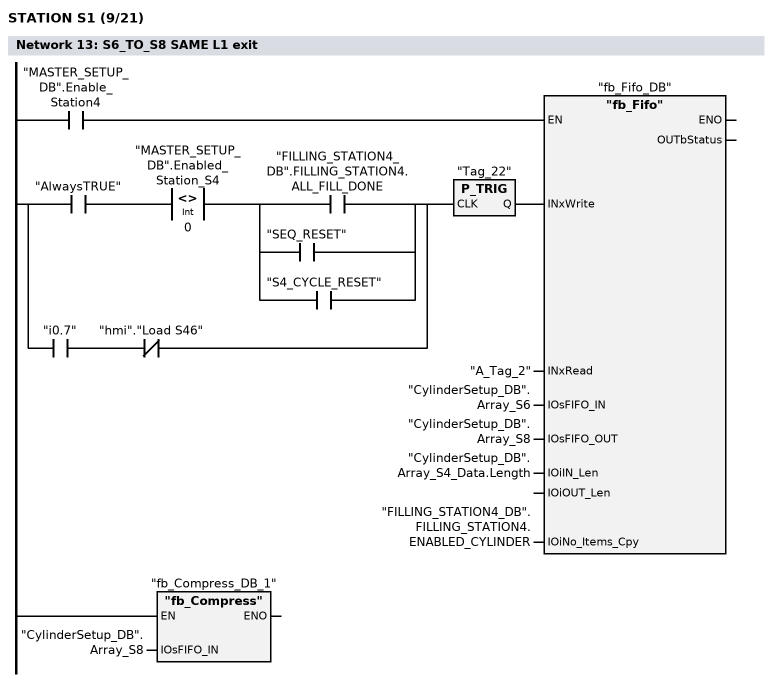
   RUNG wire#powerrail
      Contact( "MASTER_SETUP_DB".Enable_Station4 )
      "fb_Fifo_DB"(INxWrite := wire#w3, INxRead := "A_Tag_2", IOsFIFO_IN := "CylinderSetup_DB".Array_S6, IOsFIFO_OUT := "CylinderSetup_DB".Array_S8, IOiIN_Len := "CylinderSetup_DB".Array_S4_Data.Length, IOiOUT_Len :=, IOiNo_Items_Cpy := "FILLING_STATION4_DB".FILLING_STATION4.ENABLED_CYLINDER, OUTbStatus =>)
   END_RUNG
   RUNG wire#powerrail
      Contact( "AlwaysTRUE" )
      { S7_Templates := "SrcType := Int" } NE_Contact(in1 := "MASTER_SETUP_DB".Enabled_Station_S4, in2 := 0)
      wire#w1
      Contact( "FILLING_STATION4_DB".FILLING_STATION4.ALL_FILL_DONE )
      wire#w2
      P_Trig( "Tag_22" )
   END_RUNG wire#w3
   RUNG wire#w1
      Contact( "SEQ_RESET" )
   END_RUNG wire#w2
   RUNG wire#w1
      Contact( "S4_CYCLE_RESET" )
   END_RUNG wire#w2
   RUNG wire#powerrail
      Contact( "i0.7" )
      I_Contact( "hmi"."Load S46" )
   END_RUNG wire#w2
   RUNG wire#powerrail
      "fb_Compress_DB_1"(IOsFIFO_IN := "CylinderSetup_DB".Array_S8)
   END_RUNG
   // the same network as SCL:
   #_w1 := ("AlwaysTRUE" AND ("MASTER_SETUP_DB".Enabled_Station_S4 <> 0) AND ("FILLING_STATION4_DB".FILLING_STATION4.ALL_FILL_DONE OR "SEQ_RESET" OR "S4_CYCLE_RESET")) OR ("i0.7" AND NOT "hmi"."Load S46");
   #_w2 := #_w1 AND NOT "Tag_22";   // rising edge
   "Tag_22" := #_w1;
   IF "MASTER_SETUP_DB".Enable_Station4 THEN
       "fb_Fifo_DB"(INxWrite := #_w2,   // "fb_Fifo"
                    INxRead := "A_Tag_2",
                    IOsFIFO_IN := "CylinderSetup_DB".Array_S6,
                    IOsFIFO_OUT := "CylinderSetup_DB".Array_S8,
                    IOiIN_Len := "CylinderSetup_DB".Array_S4_Data.Length,
                    IOiNo_Items_Cpy := "FILLING_STATION4_DB".FILLING_STATION4.ENABLED_CYLINDER);
   END_IF;
   "fb_Compress_DB_1"(IOsFIFO_IN := "CylinderSetup_DB".Array_S8);   // "fb_Compress"
END_REGION

REGION Network 14: data move
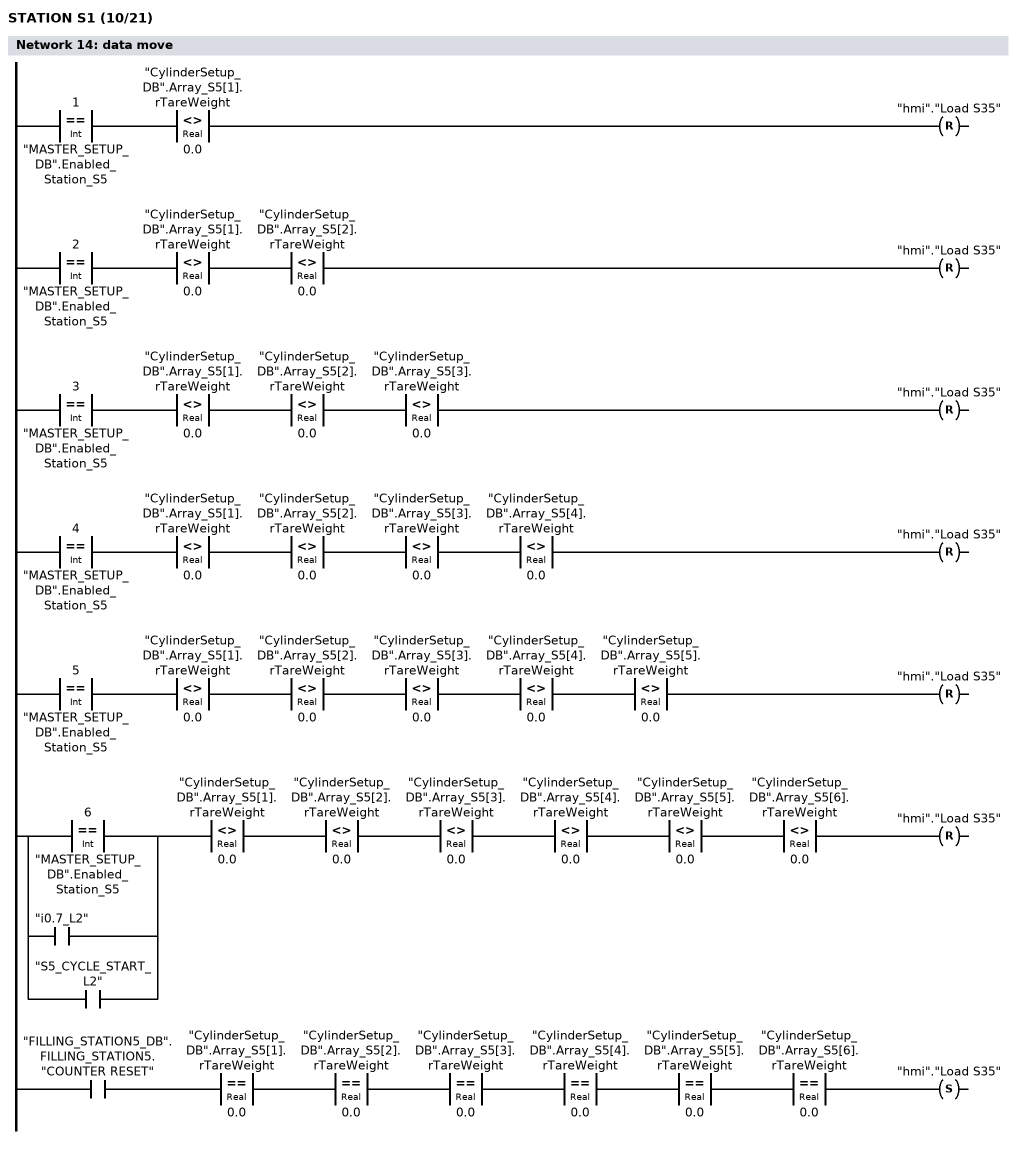
   RUNG wire#powerrail
      { S7_Templates := "SrcType := Int" } EQ_Contact(in1 := 1, in2 := "MASTER_SETUP_DB".Enabled_Station_S5)
      { S7_Templates := "SrcType := Real" } NE_Contact(in1 := "CylinderSetup_DB".Array_S5[1].rTareWeight, in2 := 0.0)
      R_Coil( "hmi"."Load S35" )
   END_RUNG
   RUNG wire#powerrail
      { S7_Templates := "SrcType := Int" } EQ_Contact(in1 := 2, in2 := "MASTER_SETUP_DB".Enabled_Station_S5)
      { S7_Templates := "SrcType := Real" } NE_Contact(in1 := "CylinderSetup_DB".Array_S5[1].rTareWeight, in2 := 0.0)
      { S7_Templates := "SrcType := Real" } NE_Contact(in1 := "CylinderSetup_DB".Array_S5[2].rTareWeight, in2 := 0.0)
      R_Coil( "hmi"."Load S35" )
   END_RUNG
   RUNG wire#powerrail
      { S7_Templates := "SrcType := Int" } EQ_Contact(in1 := 3, in2 := "MASTER_SETUP_DB".Enabled_Station_S5)
      { S7_Templates := "SrcType := Real" } NE_Contact(in1 := "CylinderSetup_DB".Array_S5[1].rTareWeight, in2 := 0.0)
      { S7_Templates := "SrcType := Real" } NE_Contact(in1 := "CylinderSetup_DB".Array_S5[2].rTareWeight, in2 := 0.0)
      { S7_Templates := "SrcType := Real" } NE_Contact(in1 := "CylinderSetup_DB".Array_S5[3].rTareWeight, in2 := 0.0)
      R_Coil( "hmi"."Load S35" )
   END_RUNG
   RUNG wire#powerrail
      { S7_Templates := "SrcType := Int" } EQ_Contact(in1 := 4, in2 := "MASTER_SETUP_DB".Enabled_Station_S5)
      { S7_Templates := "SrcType := Real" } NE_Contact(in1 := "CylinderSetup_DB".Array_S5[1].rTareWeight, in2 := 0.0)
      { S7_Templates := "SrcType := Real" } NE_Contact(in1 := "CylinderSetup_DB".Array_S5[2].rTareWeight, in2 := 0.0)
      { S7_Templates := "SrcType := Real" } NE_Contact(in1 := "CylinderSetup_DB".Array_S5[3].rTareWeight, in2 := 0.0)
      { S7_Templates := "SrcType := Real" } NE_Contact(in1 := "CylinderSetup_DB".Array_S5[4].rTareWeight, in2 := 0.0)
      R_Coil( "hmi"."Load S35" )
   END_RUNG
   RUNG wire#powerrail
      { S7_Templates := "SrcType := Int" } EQ_Contact(in1 := 5, in2 := "MASTER_SETUP_DB".Enabled_Station_S5)
      { S7_Templates := "SrcType := Real" } NE_Contact(in1 := "CylinderSetup_DB".Array_S5[1].rTareWeight, in2 := 0.0)
      { S7_Templates := "SrcType := Real" } NE_Contact(in1 := "CylinderSetup_DB".Array_S5[2].rTareWeight, in2 := 0.0)
      { S7_Templates := "SrcType := Real" } NE_Contact(in1 := "CylinderSetup_DB".Array_S5[3].rTareWeight, in2 := 0.0)
      { S7_Templates := "SrcType := Real" } NE_Contact(in1 := "CylinderSetup_DB".Array_S5[4].rTareWeight, in2 := 0.0)
      { S7_Templates := "SrcType := Real" } NE_Contact(in1 := "CylinderSetup_DB".Array_S5[5].rTareWeight, in2 := 0.0)
      R_Coil( "hmi"."Load S35" )
   END_RUNG
   RUNG wire#powerrail
      { S7_Templates := "SrcType := Int" } EQ_Contact(in1 := 6, in2 := "MASTER_SETUP_DB".Enabled_Station_S5)
      wire#w1
      { S7_Templates := "SrcType := Real" } NE_Contact(in1 := "CylinderSetup_DB".Array_S5[1].rTareWeight, in2 := 0.0)
      { S7_Templates := "SrcType := Real" } NE_Contact(in1 := "CylinderSetup_DB".Array_S5[2].rTareWeight, in2 := 0.0)
      { S7_Templates := "SrcType := Real" } NE_Contact(in1 := "CylinderSetup_DB".Array_S5[3].rTareWeight, in2 := 0.0)
      { S7_Templates := "SrcType := Real" } NE_Contact(in1 := "CylinderSetup_DB".Array_S5[4].rTareWeight, in2 := 0.0)
      { S7_Templates := "SrcType := Real" } NE_Contact(in1 := "CylinderSetup_DB".Array_S5[5].rTareWeight, in2 := 0.0)
      { S7_Templates := "SrcType := Real" } NE_Contact(in1 := "CylinderSetup_DB".Array_S5[6].rTareWeight, in2 := 0.0)
      R_Coil( "hmi"."Load S35" )
   END_RUNG
   RUNG wire#powerrail
      Contact( "i0.7_L2" )
   END_RUNG wire#w1
   RUNG wire#powerrail
      Contact( "S5_CYCLE_START_L2" )
   END_RUNG wire#w1
   RUNG wire#powerrail
      Contact( "FILLING_STATION5_DB".FILLING_STATION5."COUNTER RESET" )
      { S7_Templates := "SrcType := Real" } EQ_Contact(in1 := "CylinderSetup_DB".Array_S5[1].rTareWeight, in2 := 0.0)
      { S7_Templates := "SrcType := Real" } EQ_Contact(in1 := "CylinderSetup_DB".Array_S5[2].rTareWeight, in2 := 0.0)
      { S7_Templates := "SrcType := Real" } EQ_Contact(in1 := "CylinderSetup_DB".Array_S5[3].rTareWeight, in2 := 0.0)
      { S7_Templates := "SrcType := Real" } EQ_Contact(in1 := "CylinderSetup_DB".Array_S5[4].rTareWeight, in2 := 0.0)
      { S7_Templates := "SrcType := Real" } EQ_Contact(in1 := "CylinderSetup_DB".Array_S5[5].rTareWeight, in2 := 0.0)
      { S7_Templates := "SrcType := Real" } EQ_Contact(in1 := "CylinderSetup_DB".Array_S5[6].rTareWeight, in2 := 0.0)
      S_Coil( "hmi"."Load S35" )
   END_RUNG
   // the same network as SCL:
   IF (1 = "MASTER_SETUP_DB".Enabled_Station_S5) AND ("CylinderSetup_DB".Array_S5[1].rTareWeight <> 0.0) THEN
       "hmi"."Load S35" := FALSE;
   END_IF;
   IF (2 = "MASTER_SETUP_DB".Enabled_Station_S5) AND ("CylinderSetup_DB".Array_S5[1].rTareWeight <> 0.0) AND ("CylinderSetup_DB".Array_S5[2].rTareWeight <> 0.0) THEN
       "hmi"."Load S35" := FALSE;
   END_IF;
   IF (3 = "MASTER_SETUP_DB".Enabled_Station_S5) AND ("CylinderSetup_DB".Array_S5[1].rTareWeight <> 0.0) AND ("CylinderSetup_DB".Array_S5[2].rTareWeight <> 0.0) AND ("CylinderSetup_DB".Array_S5[3].rTareWeight <> 0.0) THEN
       "hmi"."Load S35" := FALSE;
   END_IF;
   IF (4 = "MASTER_SETUP_DB".Enabled_Station_S5) AND ("CylinderSetup_DB".Array_S5[1].rTareWeight <> 0.0) AND ("CylinderSetup_DB".Array_S5[2].rTareWeight <> 0.0) AND ("CylinderSetup_DB".Array_S5[3].rTareWeight <> 0.0) AND ("CylinderSetup_DB".Array_S5[4].rTareWeight <> 0.0) THEN
       "hmi"."Load S35" := FALSE;
   END_IF;
   IF (5 = "MASTER_SETUP_DB".Enabled_Station_S5) AND ("CylinderSetup_DB".Array_S5[1].rTareWeight <> 0.0) AND ("CylinderSetup_DB".Array_S5[2].rTareWeight <> 0.0) AND ("CylinderSetup_DB".Array_S5[3].rTareWeight <> 0.0) AND ("CylinderSetup_DB".Array_S5[4].rTareWeight <> 0.0) AND ("CylinderSetup_DB".Array_S5[5].rTareWeight <> 0.0) THEN
       "hmi"."Load S35" := FALSE;
   END_IF;
   IF ((6 = "MASTER_SETUP_DB".Enabled_Station_S5) OR "i0.7_L2" OR "S5_CYCLE_START_L2") AND ("CylinderSetup_DB".Array_S5[1].rTareWeight <> 0.0) AND ("CylinderSetup_DB".Array_S5[2].rTareWeight <> 0.0) AND ("CylinderSetup_DB".Array_S5[3].rTareWeight <> 0.0) AND ("CylinderSetup_DB".Array_S5[4].rTareWeight <> 0.0) AND ("CylinderSetup_DB".Array_S5[5].rTareWeight <> 0.0) AND ("CylinderSetup_DB".Array_S5[6].rTareWeight <> 0.0) THEN
       "hmi"."Load S35" := FALSE;
   END_IF;
   IF "FILLING_STATION5_DB".FILLING_STATION5."COUNTER RESET" AND ("CylinderSetup_DB".Array_S5[1].rTareWeight = 0.0) AND ("CylinderSetup_DB".Array_S5[2].rTareWeight = 0.0) AND ("CylinderSetup_DB".Array_S5[3].rTareWeight = 0.0) AND ("CylinderSetup_DB".Array_S5[4].rTareWeight = 0.0) AND ("CylinderSetup_DB".Array_S5[5].rTareWeight = 0.0) AND ("CylinderSetup_DB".Array_S5[6].rTareWeight = 0.0) THEN
       "hmi"."Load S35" := TRUE;
   END_IF;
END_REGION

REGION Network 15: S5_TO_S7 exit
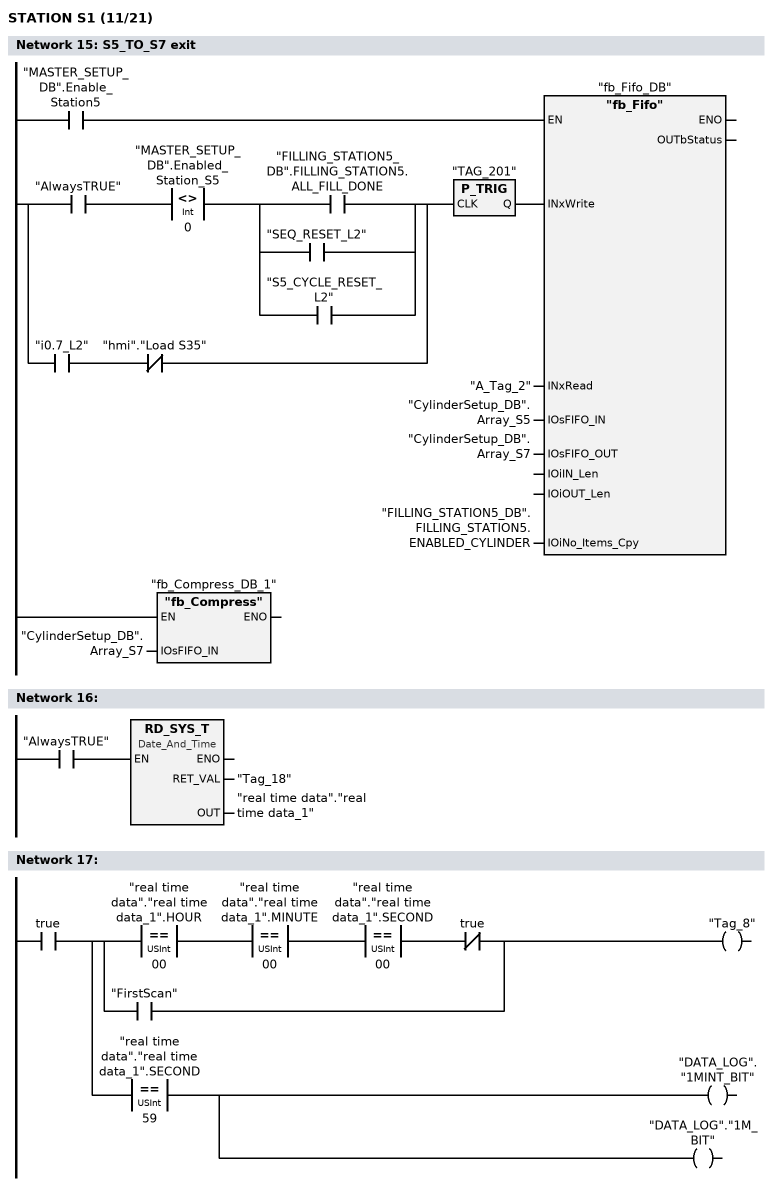
   RUNG wire#powerrail
      Contact( "MASTER_SETUP_DB".Enable_Station5 )
      "fb_Fifo_DB"(INxWrite := wire#w3, INxRead := "A_Tag_2", IOsFIFO_IN := "CylinderSetup_DB".Array_S5, IOsFIFO_OUT := "CylinderSetup_DB".Array_S7, IOiIN_Len :=, IOiOUT_Len :=, IOiNo_Items_Cpy := "FILLING_STATION5_DB".FILLING_STATION5.ENABLED_CYLINDER, OUTbStatus =>)
   END_RUNG
   RUNG wire#powerrail
      Contact( "AlwaysTRUE" )
      { S7_Templates := "SrcType := Int" } NE_Contact(in1 := "MASTER_SETUP_DB".Enabled_Station_S5, in2 := 0)
      wire#w1
      Contact( "FILLING_STATION5_DB".FILLING_STATION5.ALL_FILL_DONE )
      wire#w2
      P_Trig( "TAG_201" )
   END_RUNG wire#w3
   RUNG wire#w1
      Contact( "SEQ_RESET_L2" )
   END_RUNG wire#w2
   RUNG wire#w1
      Contact( "S5_CYCLE_RESET_L2" )
   END_RUNG wire#w2
   RUNG wire#powerrail
      Contact( "i0.7_L2" )
      I_Contact( "hmi"."Load S35" )
   END_RUNG wire#w2
   RUNG wire#powerrail
      "fb_Compress_DB_1"(IOsFIFO_IN := "CylinderSetup_DB".Array_S7)
   END_RUNG
   // the same network as SCL:
   #_w1 := ("AlwaysTRUE" AND ("MASTER_SETUP_DB".Enabled_Station_S5 <> 0) AND ("FILLING_STATION5_DB".FILLING_STATION5.ALL_FILL_DONE OR "SEQ_RESET_L2" OR "S5_CYCLE_RESET_L2")) OR ("i0.7_L2" AND NOT "hmi"."Load S35");
   #_w2 := #_w1 AND NOT "TAG_201";   // rising edge
   "TAG_201" := #_w1;
   IF "MASTER_SETUP_DB".Enable_Station5 THEN
       "fb_Fifo_DB"(INxWrite := #_w2,   // "fb_Fifo"
                    INxRead := "A_Tag_2",
                    IOsFIFO_IN := "CylinderSetup_DB".Array_S5,
                    IOsFIFO_OUT := "CylinderSetup_DB".Array_S7,
                    IOiNo_Items_Cpy := "FILLING_STATION5_DB".FILLING_STATION5.ENABLED_CYLINDER);
   END_IF;
   "fb_Compress_DB_1"(IOsFIFO_IN := "CylinderSetup_DB".Array_S7);   // "fb_Compress"
END_REGION

REGION Network 16
   RUNG wire#powerrail
      Contact( "AlwaysTRUE" )
      { S7_Templates := "date_type := Date_And_Time" } RD_SYS_T(RET_VAL => "Tag_18", OUT => "real time data"."real time data_1")
   END_RUNG
   // the same network as SCL:
   IF "AlwaysTRUE" THEN "Tag_18" := RD_SYS_T(OUT => "real time data"."real time data_1"); END_IF;
END_REGION

REGION Network 17
   RUNG wire#powerrail
      Contact( true )
      wire#w1
      { S7_Templates := "SrcType := USInt" } EQ_Contact(in1 := "real time data"."real time data_1".HOUR, in2 := 00)
      { S7_Templates := "SrcType := USInt" } EQ_Contact(in1 := "real time data"."real time data_1".MINUTE, in2 := 00)
      { S7_Templates := "SrcType := USInt" } EQ_Contact(in1 := "real time data"."real time data_1".SECOND, in2 := 00)
      I_Contact( true )
      wire#w2
      Coil( "Tag_8" )
   END_RUNG
   RUNG wire#w1
      Contact( "FirstScan" )
   END_RUNG wire#w2
   RUNG wire#w1
      { S7_Templates := "SrcType := USInt" } EQ_Contact(in1 := "real time data"."real time data_1".SECOND, in2 := 59)
      wire#w3
      Coil( "DATA_LOG"."1MINT_BIT" )
   END_RUNG
   RUNG wire#w3
      Coil( "DATA_LOG"."1M_BIT" )
   END_RUNG
   // the same network as SCL:
   "Tag_8" := true AND ((("real time data"."real time data_1".HOUR = 00) AND ("real time data"."real time data_1".MINUTE = 00) AND ("real time data"."real time data_1".SECOND = 00) AND NOT true) OR "FirstScan");
   "DATA_LOG"."1MINT_BIT" := true AND ("real time data"."real time data_1".SECOND = 59);
   "DATA_LOG"."1M_BIT" := "DATA_LOG"."1MINT_BIT";
END_REGION

REGION Network 18 (SCL): S4 S6 FIFO DATA SKIP
   #idx2 := 0;
   #idx3 := 0;

   IF "AlwaysTRUE" THEN
       FOR #idx2 := 1 TO "MASTER_SETUP_DB".S4_Total_Station DO

           IF "MASTER_SETUP_DB".S4_Enabled_Station[#idx2]  THEN
               #idx3 := #idx3 + 1;
               "hmi_dummy_array".S4_PrefillingDummyData[#idx2] := "CylinderSetup_DB".Array_S6[#idx3];

             ELSIF
                #idx2 > "MASTER_SETUP_DB".S4_Total_Station OR #idx3 >"MASTER_SETUP_DB".S4_Total_Station THEN
                   EXIT;
               END_IF;
           END_FOR;


   END_IF;
END_REGION

REGION Network 19 (SCL)
   #idx4 := 0;
   #idx6 := 0;

   IF "AlwaysTRUE" THEN
       FOR #idx4 := 1 TO "MASTER_SETUP_DB".S5_Total_Station DO

           IF "MASTER_SETUP_DB".S5_Enabled_Station[#idx4] THEN
               #idx6 := #idx6 + 1;
               "hmi_dummy_array".S5_PrefillingdummyData[#idx4] := "CylinderSetup_DB".Array_S5[#idx6];

           ELSIF
               #idx4 > "MASTER_SETUP_DB".S5_Total_Station OR #idx6 > "MASTER_SETUP_DB".S5_Total_Station THEN
               EXIT;
           END_IF;
       END_FOR;


   END_IF;
END_REGION

REGION Network 20
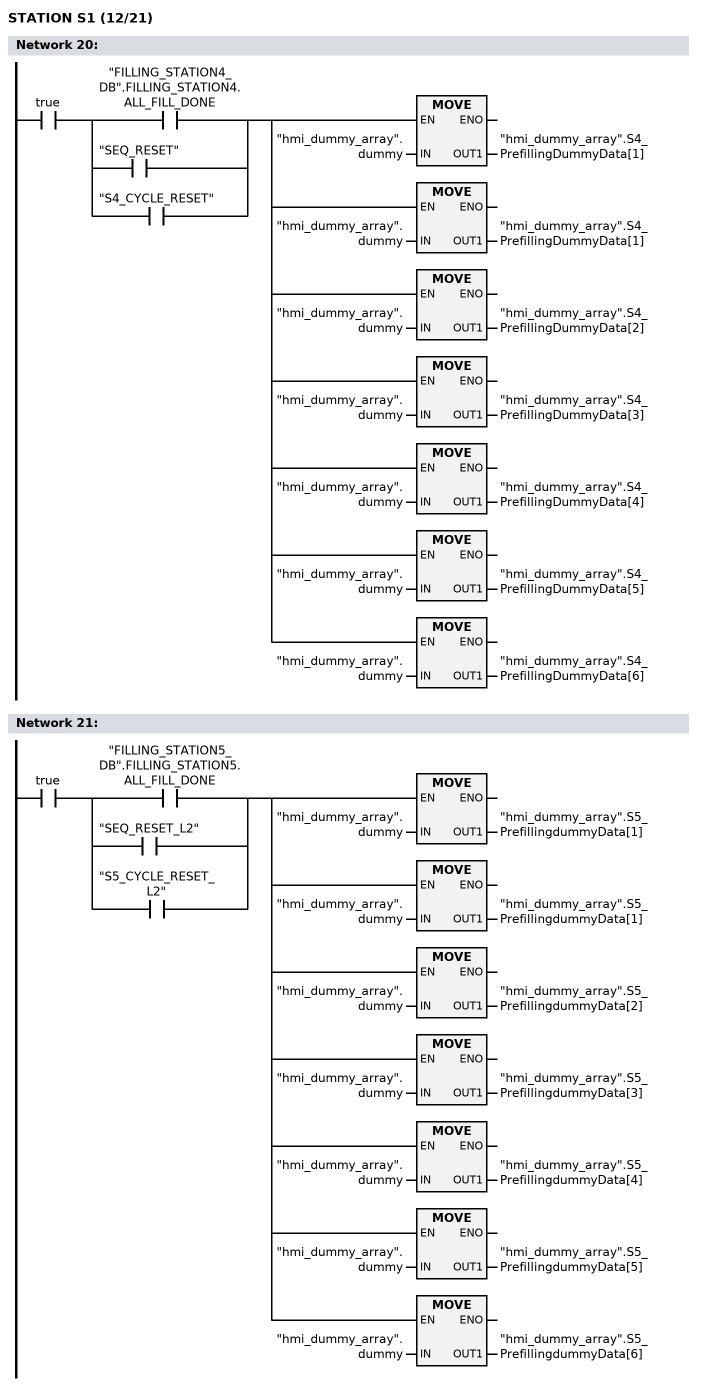
   RUNG wire#powerrail
      Contact( true )
      wire#w1
      Contact( "FILLING_STATION4_DB".FILLING_STATION4.ALL_FILL_DONE )
      wire#w2
      Move(in := "hmi_dummy_array".dummy, out1 => "hmi_dummy_array".S4_PrefillingDummyData[1])
   END_RUNG
   RUNG wire#w1
      Contact( "SEQ_RESET" )
   END_RUNG wire#w2
   RUNG wire#w1
      Contact( "S4_CYCLE_RESET" )
   END_RUNG wire#w2
   RUNG wire#w2
      Move(in := "hmi_dummy_array".dummy, out1 => "hmi_dummy_array".S4_PrefillingDummyData[1])
   END_RUNG
   RUNG wire#w2
      Move(in := "hmi_dummy_array".dummy, out1 => "hmi_dummy_array".S4_PrefillingDummyData[2])
   END_RUNG
   RUNG wire#w2
      Move(in := "hmi_dummy_array".dummy, out1 => "hmi_dummy_array".S4_PrefillingDummyData[3])
   END_RUNG
   RUNG wire#w2
      Move(in := "hmi_dummy_array".dummy, out1 => "hmi_dummy_array".S4_PrefillingDummyData[4])
   END_RUNG
   RUNG wire#w2
      Move(in := "hmi_dummy_array".dummy, out1 => "hmi_dummy_array".S4_PrefillingDummyData[5])
   END_RUNG
   RUNG wire#w2
      Move(in := "hmi_dummy_array".dummy, out1 => "hmi_dummy_array".S4_PrefillingDummyData[6])
   END_RUNG
   // the same network as SCL:
   IF true AND ("FILLING_STATION4_DB".FILLING_STATION4.ALL_FILL_DONE OR "SEQ_RESET" OR "S4_CYCLE_RESET") THEN
       "hmi_dummy_array".S4_PrefillingDummyData[1] := "hmi_dummy_array".dummy;
       "hmi_dummy_array".S4_PrefillingDummyData[1] := "hmi_dummy_array".dummy;
       "hmi_dummy_array".S4_PrefillingDummyData[2] := "hmi_dummy_array".dummy;
       "hmi_dummy_array".S4_PrefillingDummyData[3] := "hmi_dummy_array".dummy;
       "hmi_dummy_array".S4_PrefillingDummyData[4] := "hmi_dummy_array".dummy;
       "hmi_dummy_array".S4_PrefillingDummyData[5] := "hmi_dummy_array".dummy;
       "hmi_dummy_array".S4_PrefillingDummyData[6] := "hmi_dummy_array".dummy;
   END_IF;
END_REGION

REGION Network 21
   RUNG wire#powerrail
      Contact( true )
      wire#w1
      Contact( "FILLING_STATION5_DB".FILLING_STATION5.ALL_FILL_DONE )
      wire#w2
      Move(in := "hmi_dummy_array".dummy, out1 => "hmi_dummy_array".S5_PrefillingdummyData[1])
   END_RUNG
   RUNG wire#w1
      Contact( "SEQ_RESET_L2" )
   END_RUNG wire#w2
   RUNG wire#w1
      Contact( "S5_CYCLE_RESET_L2" )
   END_RUNG wire#w2
   RUNG wire#w2
      Move(in := "hmi_dummy_array".dummy, out1 => "hmi_dummy_array".S5_PrefillingdummyData[1])
   END_RUNG
   RUNG wire#w2
      Move(in := "hmi_dummy_array".dummy, out1 => "hmi_dummy_array".S5_PrefillingdummyData[2])
   END_RUNG
   RUNG wire#w2
      Move(in := "hmi_dummy_array".dummy, out1 => "hmi_dummy_array".S5_PrefillingdummyData[3])
   END_RUNG
   RUNG wire#w2
      Move(in := "hmi_dummy_array".dummy, out1 => "hmi_dummy_array".S5_PrefillingdummyData[4])
   END_RUNG
   RUNG wire#w2
      Move(in := "hmi_dummy_array".dummy, out1 => "hmi_dummy_array".S5_PrefillingdummyData[5])
   END_RUNG
   RUNG wire#w2
      Move(in := "hmi_dummy_array".dummy, out1 => "hmi_dummy_array".S5_PrefillingdummyData[6])
   END_RUNG
   // the same network as SCL:
   IF true AND ("FILLING_STATION5_DB".FILLING_STATION5.ALL_FILL_DONE OR "SEQ_RESET_L2" OR "S5_CYCLE_RESET_L2") THEN
       "hmi_dummy_array".S5_PrefillingdummyData[1] := "hmi_dummy_array".dummy;
       "hmi_dummy_array".S5_PrefillingdummyData[1] := "hmi_dummy_array".dummy;
       "hmi_dummy_array".S5_PrefillingdummyData[2] := "hmi_dummy_array".dummy;
       "hmi_dummy_array".S5_PrefillingdummyData[3] := "hmi_dummy_array".dummy;
       "hmi_dummy_array".S5_PrefillingdummyData[4] := "hmi_dummy_array".dummy;
       "hmi_dummy_array".S5_PrefillingdummyData[5] := "hmi_dummy_array".dummy;
       "hmi_dummy_array".S5_PrefillingdummyData[6] := "hmi_dummy_array".dummy;
   END_IF;
END_REGION

REGION Network 22
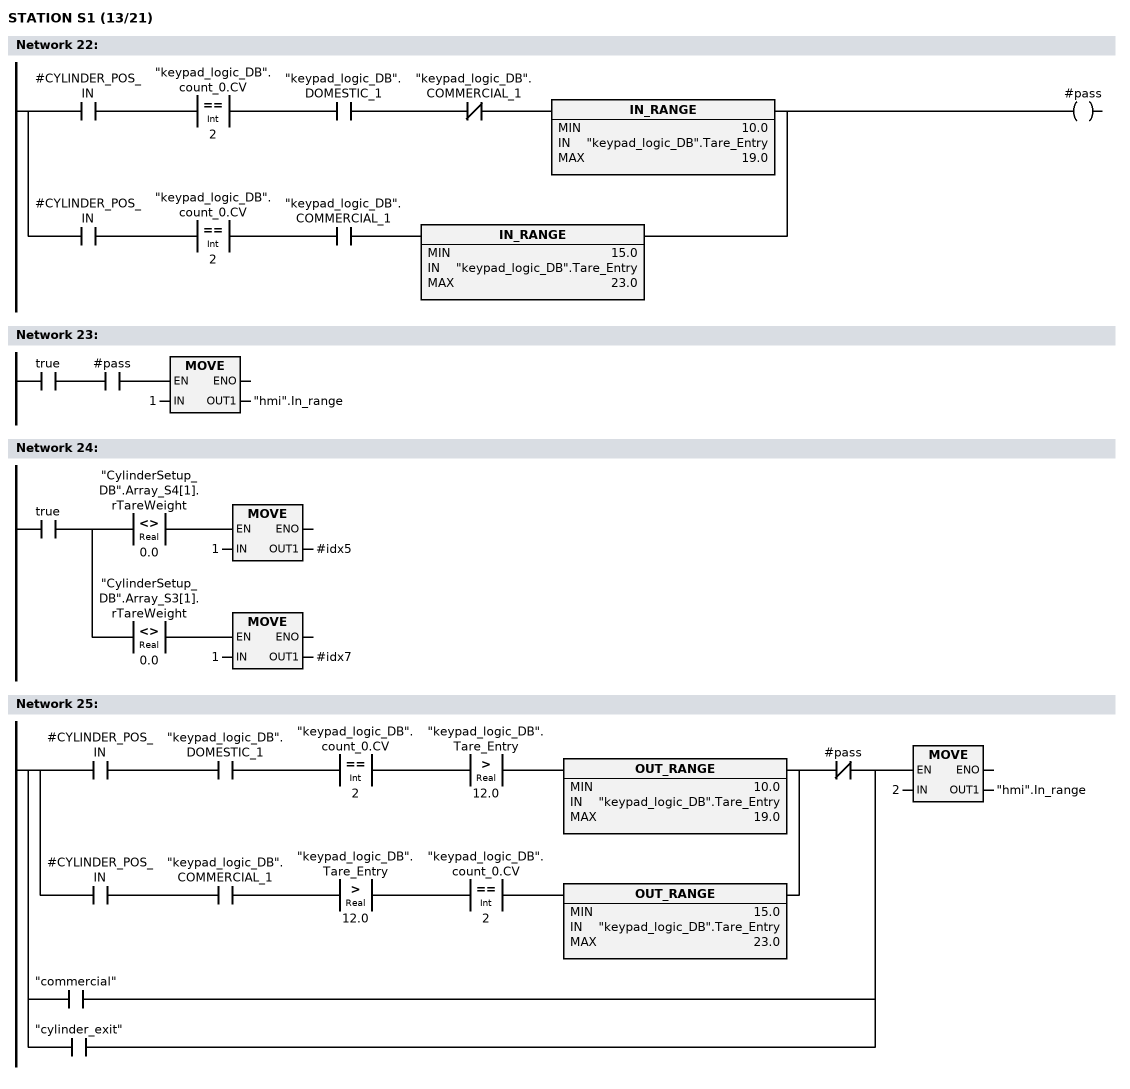
   RUNG wire#powerrail
      Contact( #CYLINDER_POS_IN )
      { S7_Templates := "SrcType := Int" } EQ_Contact(in1 := "keypad_logic_DB".count_0.CV, in2 := 2)
      Contact( "keypad_logic_DB".DOMESTIC_1 )
      I_Contact( "keypad_logic_DB".COMMERCIAL_1 )
      { S7_Templates := "SrcType := Real" } InRange(min := 10.0, in := "keypad_logic_DB".Tare_Entry, max := 19.0)
      wire#w1
      Coil( #pass )
   END_RUNG
   RUNG wire#powerrail
      Contact( #CYLINDER_POS_IN )
      { S7_Templates := "SrcType := Int" } EQ_Contact(in1 := "keypad_logic_DB".count_0.CV, in2 := 2)
      Contact( "keypad_logic_DB".COMMERCIAL_1 )
      { S7_Templates := "SrcType := Real" } InRange(min := 15.0, in := "keypad_logic_DB".Tare_Entry, max := 23.0)
   END_RUNG wire#w1
   // the same network as SCL:
   #pass := (#CYLINDER_POS_IN AND ("keypad_logic_DB".count_0.CV = 2) AND "keypad_logic_DB".DOMESTIC_1 AND NOT "keypad_logic_DB".COMMERCIAL_1 AND (10.0 <= "keypad_logic_DB".Tare_Entry) AND ("keypad_logic_DB".Tare_Entry <= 19.0)) OR (#CYLINDER_POS_IN AND ("keypad_logic_DB".count_0.CV = 2) AND "keypad_logic_DB".COMMERCIAL_1 AND (15.0 <= "keypad_logic_DB".Tare_Entry) AND ("keypad_logic_DB".Tare_Entry <= 23.0));
END_REGION

REGION Network 23
   RUNG wire#powerrail
      Contact( true )
      Contact( #pass )
      Move(in := 1, out1 => "hmi".In_range)
   END_RUNG
   // the same network as SCL:
   IF true AND #pass THEN "hmi".In_range := 1; END_IF;
END_REGION

REGION Network 24
   RUNG wire#powerrail
      Contact( true )
      wire#w1
      { S7_Templates := "SrcType := Real" } NE_Contact(in1 := "CylinderSetup_DB".Array_S4[1].rTareWeight, in2 := 0.0)
      Move(in := 1, out1 => #idx5)
   END_RUNG
   RUNG wire#w1
      { S7_Templates := "SrcType := Real" } NE_Contact(in1 := "CylinderSetup_DB".Array_S3[1].rTareWeight, in2 := 0.0)
      Move(in := 1, out1 => #idx7)
   END_RUNG
   // the same network as SCL:
   IF true AND ("CylinderSetup_DB".Array_S4[1].rTareWeight <> 0.0) THEN #idx5 := 1; END_IF;
   IF true AND ("CylinderSetup_DB".Array_S3[1].rTareWeight <> 0.0) THEN #idx7 := 1; END_IF;
END_REGION

REGION Network 25
   IF (((#CYLINDER_POS_IN AND "keypad_logic_DB".DOMESTIC_1 AND ("keypad_logic_DB".count_0.CV = 2) AND ("keypad_logic_DB".Tare_Entry > 12.0) AND (("keypad_logic_DB".Tare_Entry < 10.0) OR ("keypad_logic_DB".Tare_Entry > 19.0))) OR (#CYLINDER_POS_IN AND "keypad_logic_DB".COMMERCIAL_1 AND ("keypad_logic_DB".Tare_Entry > 12.0) AND ("keypad_logic_DB".count_0.CV = 2) AND (("keypad_logic_DB".Tare_Entry < 15.0) OR ("keypad_logic_DB".Tare_Entry > 23.0)))) AND NOT #pass) OR "commercial" OR "cylinder_exit" THEN
       "hmi".In_range := 2;
   END_IF;
END_REGION

REGION Network 26
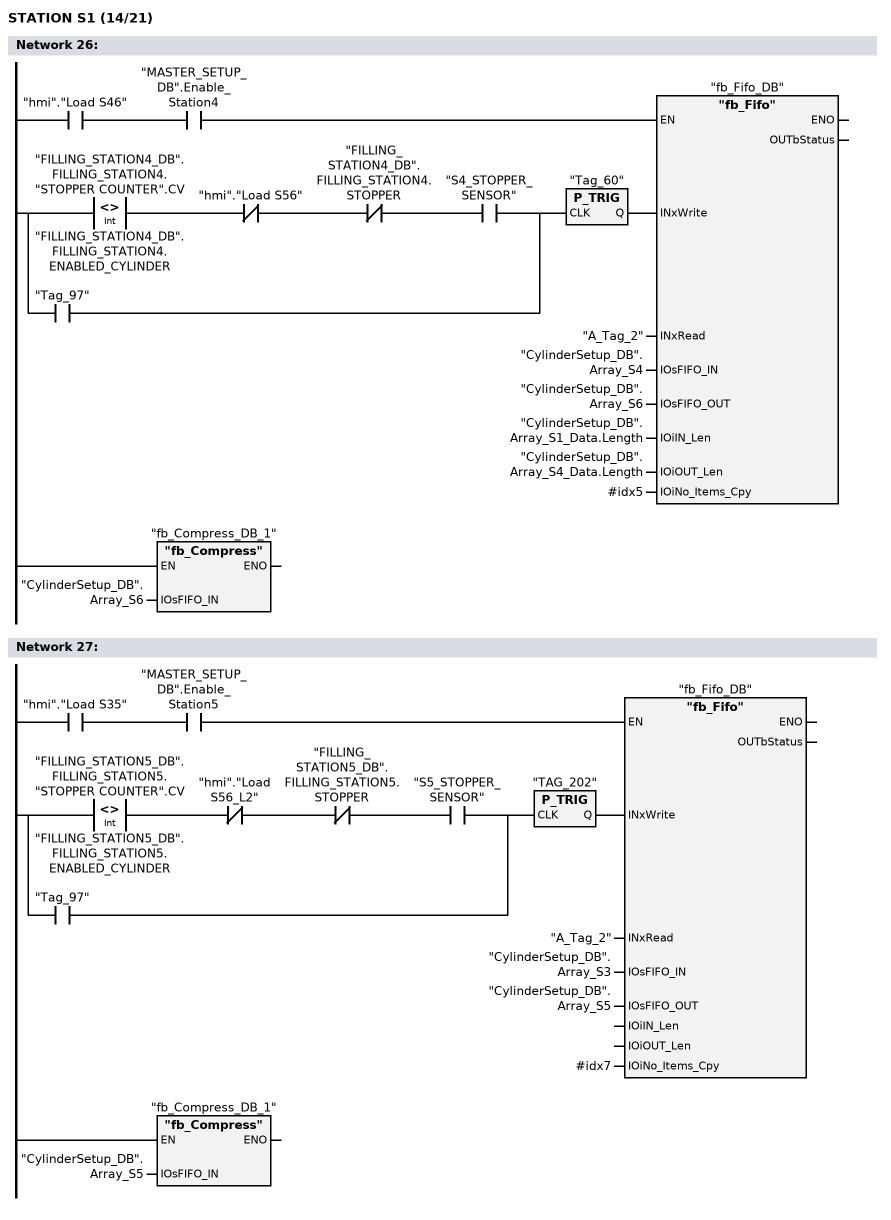
   RUNG wire#powerrail
      Contact( "hmi"."Load S46" )
      Contact( "MASTER_SETUP_DB".Enable_Station4 )
      "fb_Fifo_DB"(INxWrite := wire#w2, INxRead := "A_Tag_2", IOsFIFO_IN := "CylinderSetup_DB".Array_S4, IOsFIFO_OUT := "CylinderSetup_DB".Array_S6, IOiIN_Len := "CylinderSetup_DB".Array_S1_Data.Length, IOiOUT_Len := "CylinderSetup_DB".Array_S4_Data.Length, IOiNo_Items_Cpy := #idx5, OUTbStatus =>)
   END_RUNG
   RUNG wire#powerrail
      { S7_Templates := "SrcType := Int" } NE_Contact(in1 := "FILLING_STATION4_DB".FILLING_STATION4."STOPPER COUNTER".CV, in2 := "FILLING_STATION4_DB".FILLING_STATION4.ENABLED_CYLINDER)
      I_Contact( "hmi"."Load S56" )
      I_Contact( "FILLING_STATION4_DB".FILLING_STATION4.STOPPER )
      Contact( "S4_STOPPER_SENSOR" )
      wire#w1
      P_Trig( "Tag_60" )
   END_RUNG wire#w2
   RUNG wire#powerrail
      Contact( "Tag_97" )
   END_RUNG wire#w1
   RUNG wire#powerrail
      "fb_Compress_DB_1"(IOsFIFO_IN := "CylinderSetup_DB".Array_S6)
   END_RUNG
   // the same network as SCL:
   #_w1 := (("FILLING_STATION4_DB".FILLING_STATION4."STOPPER COUNTER".CV <> "FILLING_STATION4_DB".FILLING_STATION4.ENABLED_CYLINDER) AND NOT "hmi"."Load S56" AND NOT "FILLING_STATION4_DB".FILLING_STATION4.STOPPER AND "S4_STOPPER_SENSOR") OR "Tag_97";
   #_w2 := #_w1 AND NOT "Tag_60";   // rising edge
   "Tag_60" := #_w1;
   IF "hmi"."Load S46" AND "MASTER_SETUP_DB".Enable_Station4 THEN
       "fb_Fifo_DB"(INxWrite := #_w2,   // "fb_Fifo"
                    INxRead := "A_Tag_2",
                    IOsFIFO_IN := "CylinderSetup_DB".Array_S4,
                    IOsFIFO_OUT := "CylinderSetup_DB".Array_S6,
                    IOiIN_Len := "CylinderSetup_DB".Array_S1_Data.Length,
                    IOiOUT_Len := "CylinderSetup_DB".Array_S4_Data.Length,
                    IOiNo_Items_Cpy := #idx5);
   END_IF;
   "fb_Compress_DB_1"(IOsFIFO_IN := "CylinderSetup_DB".Array_S6);   // "fb_Compress"
END_REGION

REGION Network 27
   RUNG wire#powerrail
      Contact( "hmi"."Load S35" )
      Contact( "MASTER_SETUP_DB".Enable_Station5 )
      "fb_Fifo_DB"(INxWrite := wire#w2, INxRead := "A_Tag_2", IOsFIFO_IN := "CylinderSetup_DB".Array_S3, IOsFIFO_OUT := "CylinderSetup_DB".Array_S5, IOiIN_Len :=, IOiOUT_Len :=, IOiNo_Items_Cpy := #idx7, OUTbStatus =>)
   END_RUNG
   RUNG wire#powerrail
      { S7_Templates := "SrcType := Int" } NE_Contact(in1 := "FILLING_STATION5_DB".FILLING_STATION5."STOPPER COUNTER".CV, in2 := "FILLING_STATION5_DB".FILLING_STATION5.ENABLED_CYLINDER)
      I_Contact( "hmi"."Load S56_L2" )
      I_Contact( "FILLING_STATION5_DB".FILLING_STATION5.STOPPER )
      Contact( "S5_STOPPER_SENSOR" )
      wire#w1
      P_Trig( "TAG_202" )
   END_RUNG wire#w2
   RUNG wire#powerrail
      Contact( "Tag_97" )
   END_RUNG wire#w1
   RUNG wire#powerrail
      "fb_Compress_DB_1"(IOsFIFO_IN := "CylinderSetup_DB".Array_S5)
   END_RUNG
   // the same network as SCL:
   #_w1 := (("FILLING_STATION5_DB".FILLING_STATION5."STOPPER COUNTER".CV <> "FILLING_STATION5_DB".FILLING_STATION5.ENABLED_CYLINDER) AND NOT "hmi"."Load S56_L2" AND NOT "FILLING_STATION5_DB".FILLING_STATION5.STOPPER AND "S5_STOPPER_SENSOR") OR "Tag_97";
   #_w2 := #_w1 AND NOT "TAG_202";   // rising edge
   "TAG_202" := #_w1;
   IF "hmi"."Load S35" AND "MASTER_SETUP_DB".Enable_Station5 THEN
       "fb_Fifo_DB"(INxWrite := #_w2,   // "fb_Fifo"
                    INxRead := "A_Tag_2",
                    IOsFIFO_IN := "CylinderSetup_DB".Array_S3,
                    IOsFIFO_OUT := "CylinderSetup_DB".Array_S5,
                    IOiNo_Items_Cpy := #idx7);
   END_IF;
   "fb_Compress_DB_1"(IOsFIFO_IN := "CylinderSetup_DB".Array_S5);   // "fb_Compress"
END_REGION

REGION Network 28
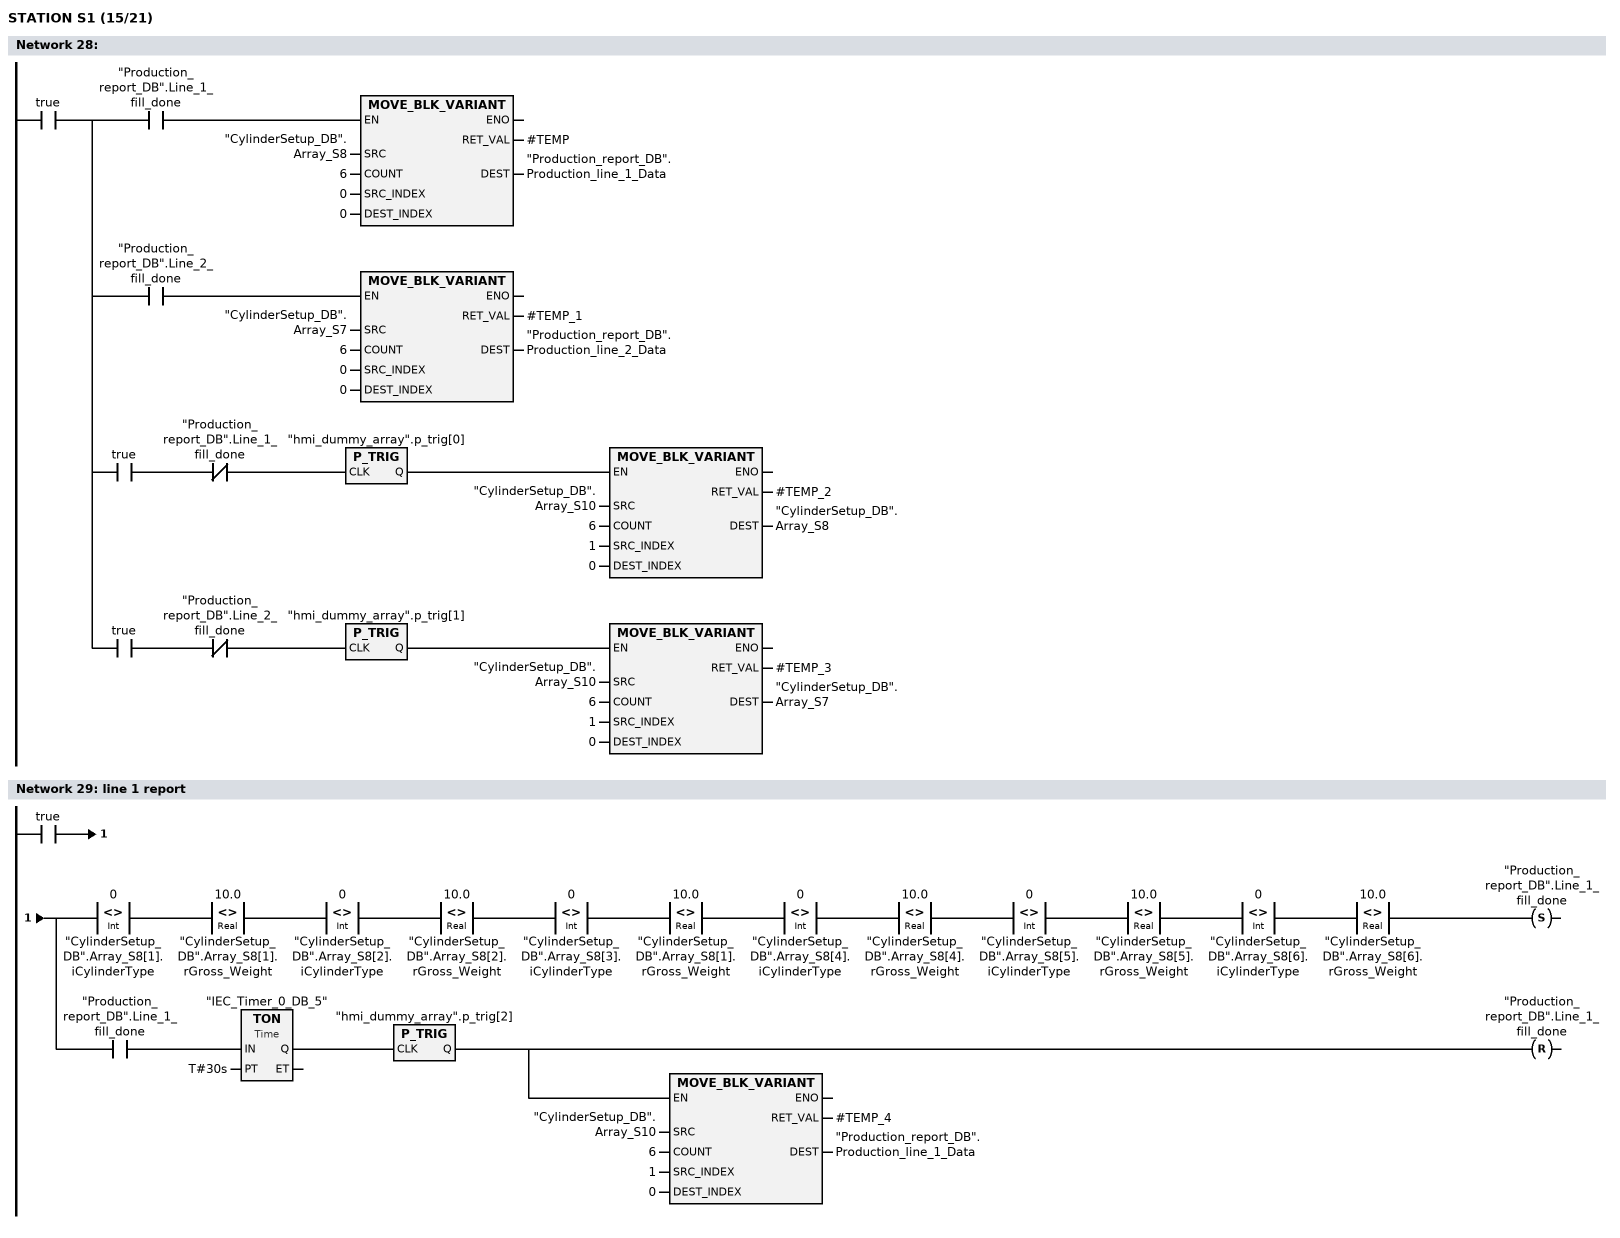
   RUNG wire#powerrail
      Contact( true )
      wire#w1
      Contact( "Production_report_DB".Line_1_fill_done )
      MOVE_BLK_VARIANT(SRC := "CylinderSetup_DB".Array_S8, COUNT := 6, SRC_INDEX := 0, DEST_INDEX := 0, Ret_Val => #TEMP, DEST => "Production_report_DB".Production_line_1_Data)
   END_RUNG
   RUNG wire#w1
      Contact( "Production_report_DB".Line_2_fill_done )
      MOVE_BLK_VARIANT(SRC := "CylinderSetup_DB".Array_S7, COUNT := 6, SRC_INDEX := 0, DEST_INDEX := 0, Ret_Val => #TEMP_1, DEST => "Production_report_DB".Production_line_2_Data)
   END_RUNG
   RUNG wire#w1
      Contact( true )
      I_Contact( "Production_report_DB".Line_1_fill_done )
      P_Trig( "hmi_dummy_array".p_trig[0] )
      MOVE_BLK_VARIANT(SRC := "CylinderSetup_DB".Array_S10, COUNT := 6, SRC_INDEX := 1, DEST_INDEX := 0, Ret_Val => #TEMP_2, DEST => "CylinderSetup_DB".Array_S8)
   END_RUNG
   RUNG wire#w1
      Contact( true )
      I_Contact( "Production_report_DB".Line_2_fill_done )
      P_Trig( "hmi_dummy_array".p_trig[1] )
      MOVE_BLK_VARIANT(SRC := "CylinderSetup_DB".Array_S10, COUNT := 6, SRC_INDEX := 1, DEST_INDEX := 0, Ret_Val => #TEMP_3, DEST => "CylinderSetup_DB".Array_S7)
   END_RUNG
   // the same network as SCL:
   IF true AND "Production_report_DB".Line_1_fill_done THEN
       #TEMP := MOVE_BLK_VARIANT(SRC := "CylinderSetup_DB".Array_S8,
                               COUNT := 6,
                               SRC_INDEX := 0,
                               DEST_INDEX := 0,
                               DEST => "Production_report_DB".Production_line_1_Data);
   END_IF;
   IF true AND "Production_report_DB".Line_2_fill_done THEN
       #TEMP_1 := MOVE_BLK_VARIANT(SRC := "CylinderSetup_DB".Array_S7,
                               COUNT := 6,
                               SRC_INDEX := 0,
                               DEST_INDEX := 0,
                               DEST => "Production_report_DB".Production_line_2_Data);
   END_IF;
   #_w1 := true AND true AND NOT "Production_report_DB".Line_1_fill_done;
   #_w2 := #_w1 AND NOT "hmi_dummy_array".p_trig[0];   // rising edge
   "hmi_dummy_array".p_trig[0] := #_w1;
   IF #_w2 THEN
       #TEMP_2 := MOVE_BLK_VARIANT(SRC := "CylinderSetup_DB".Array_S10,
                               COUNT := 6,
                               SRC_INDEX := 1,
                               DEST_INDEX := 0,
                               DEST => "CylinderSetup_DB".Array_S8);
   END_IF;
   #_w3 := true AND true AND NOT "Production_report_DB".Line_2_fill_done;
   #_w4 := #_w3 AND NOT "hmi_dummy_array".p_trig[1];   // rising edge
   "hmi_dummy_array".p_trig[1] := #_w3;
   IF #_w4 THEN
       #TEMP_3 := MOVE_BLK_VARIANT(SRC := "CylinderSetup_DB".Array_S10,
                               COUNT := 6,
                               SRC_INDEX := 1,
                               DEST_INDEX := 0,
                               DEST => "CylinderSetup_DB".Array_S7);
   END_IF;
END_REGION

REGION Network 29: line 1 report
   RUNG wire#powerrail
      Contact( true )
      wire#w1
      { S7_Templates := "SrcType := Int" } NE_Contact(in1 := 0, in2 := "CylinderSetup_DB".Array_S8[1].iCylinderType)
      { S7_Templates := "SrcType := Real" } NE_Contact(in1 := 10.0, in2 := "CylinderSetup_DB".Array_S8[1].rGross_Weight)
      { S7_Templates := "SrcType := Int" } NE_Contact(in1 := 0, in2 := "CylinderSetup_DB".Array_S8[2].iCylinderType)
      { S7_Templates := "SrcType := Real" } NE_Contact(in1 := 10.0, in2 := "CylinderSetup_DB".Array_S8[2].rGross_Weight)
      { S7_Templates := "SrcType := Int" } NE_Contact(in1 := 0, in2 := "CylinderSetup_DB".Array_S8[3].iCylinderType)
      { S7_Templates := "SrcType := Real" } NE_Contact(in1 := 10.0, in2 := "CylinderSetup_DB".Array_S8[1].rGross_Weight)
      { S7_Templates := "SrcType := Int" } NE_Contact(in1 := 0, in2 := "CylinderSetup_DB".Array_S8[4].iCylinderType)
      { S7_Templates := "SrcType := Real" } NE_Contact(in1 := 10.0, in2 := "CylinderSetup_DB".Array_S8[4].rGross_Weight)
      { S7_Templates := "SrcType := Int" } NE_Contact(in1 := 0, in2 := "CylinderSetup_DB".Array_S8[5].iCylinderType)
      { S7_Templates := "SrcType := Real" } NE_Contact(in1 := 10.0, in2 := "CylinderSetup_DB".Array_S8[5].rGross_Weight)
      { S7_Templates := "SrcType := Int" } NE_Contact(in1 := 0, in2 := "CylinderSetup_DB".Array_S8[6].iCylinderType)
      { S7_Templates := "SrcType := Real" } NE_Contact(in1 := 10.0, in2 := "CylinderSetup_DB".Array_S8[6].rGross_Weight)
      S_Coil( "Production_report_DB".Line_1_fill_done )
   END_RUNG
   RUNG wire#w1
      Contact( "Production_report_DB".Line_1_fill_done )
      { S7_Templates := "time_type := Time" } "IEC_Timer_0_DB_5".TON(pt := T#30s, et =>)
      P_Trig( "hmi_dummy_array".p_trig[2] )
      wire#w2
      R_Coil( "Production_report_DB".Line_1_fill_done )
   END_RUNG
   RUNG wire#w2
      MOVE_BLK_VARIANT(SRC := "CylinderSetup_DB".Array_S10, COUNT := 6, SRC_INDEX := 1, DEST_INDEX := 0, Ret_Val => #TEMP_4, DEST => "Production_report_DB".Production_line_1_Data)
   END_RUNG
   // the same network as SCL:
   IF true AND (0 <> "CylinderSetup_DB".Array_S8[1].iCylinderType) AND (10.0 <> "CylinderSetup_DB".Array_S8[1].rGross_Weight) AND (0 <> "CylinderSetup_DB".Array_S8[2].iCylinderType) AND (10.0 <> "CylinderSetup_DB".Array_S8[2].rGross_Weight) AND (0 <> "CylinderSetup_DB".Array_S8[3].iCylinderType) AND (10.0 <> "CylinderSetup_DB".Array_S8[1].rGross_Weight) AND (0 <> "CylinderSetup_DB".Array_S8[4].iCylinderType) AND (10.0 <> "CylinderSetup_DB".Array_S8[4].rGross_Weight) AND (0 <> "CylinderSetup_DB".Array_S8[5].iCylinderType) AND (10.0 <> "CylinderSetup_DB".Array_S8[5].rGross_Weight) AND (0 <> "CylinderSetup_DB".Array_S8[6].iCylinderType) AND (10.0 <> "CylinderSetup_DB".Array_S8[6].rGross_Weight) THEN
       "Production_report_DB".Line_1_fill_done := TRUE;
   END_IF;
   "IEC_Timer_0_DB_5".TON(IN := true AND "Production_report_DB".Line_1_fill_done, PT := T#30s);
   #_w1 := "IEC_Timer_0_DB_5".Q AND NOT "hmi_dummy_array".p_trig[2];   // rising edge
   "hmi_dummy_array".p_trig[2] := "IEC_Timer_0_DB_5".Q;
   IF #_w1 THEN
       "Production_report_DB".Line_1_fill_done := FALSE;
       #TEMP_4 := MOVE_BLK_VARIANT(SRC := "CylinderSetup_DB".Array_S10,
                               COUNT := 6,
                               SRC_INDEX := 1,
                               DEST_INDEX := 0,
                               DEST => "Production_report_DB".Production_line_1_Data);
   END_IF;
END_REGION

REGION Network 30: line 2 report
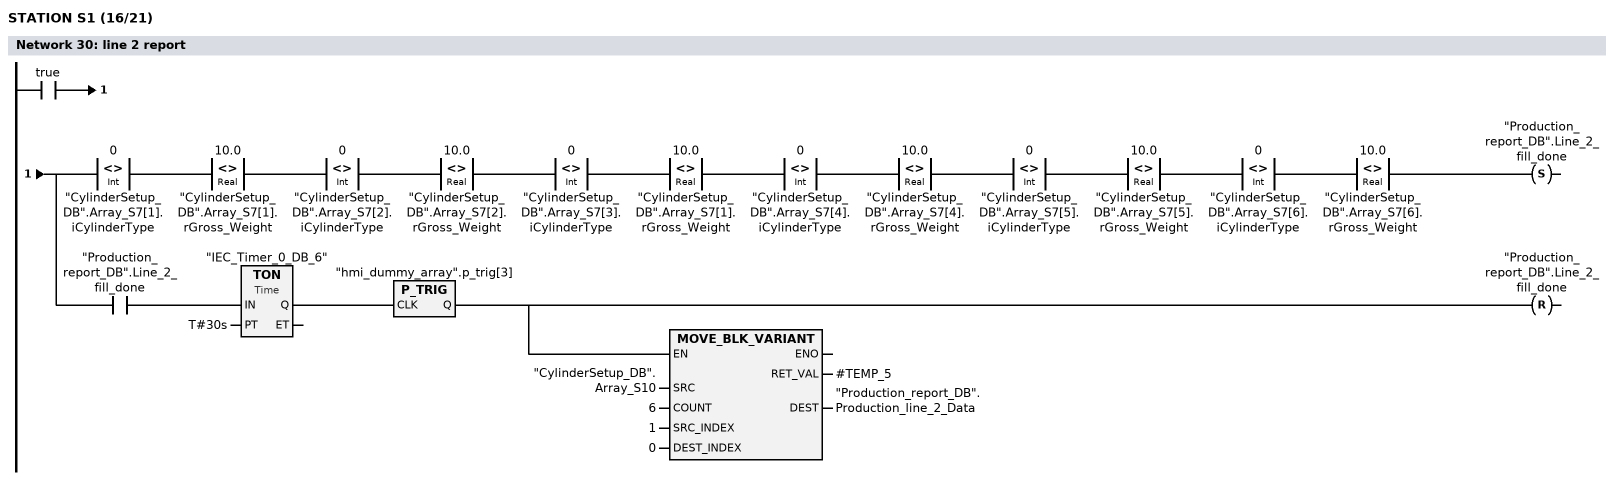
   RUNG wire#powerrail
      Contact( true )
      wire#w1
      { S7_Templates := "SrcType := Int" } NE_Contact(in1 := 0, in2 := "CylinderSetup_DB".Array_S7[1].iCylinderType)
      { S7_Templates := "SrcType := Real" } NE_Contact(in1 := 10.0, in2 := "CylinderSetup_DB".Array_S7[1].rGross_Weight)
      { S7_Templates := "SrcType := Int" } NE_Contact(in1 := 0, in2 := "CylinderSetup_DB".Array_S7[2].iCylinderType)
      { S7_Templates := "SrcType := Real" } NE_Contact(in1 := 10.0, in2 := "CylinderSetup_DB".Array_S7[2].rGross_Weight)
      { S7_Templates := "SrcType := Int" } NE_Contact(in1 := 0, in2 := "CylinderSetup_DB".Array_S7[3].iCylinderType)
      { S7_Templates := "SrcType := Real" } NE_Contact(in1 := 10.0, in2 := "CylinderSetup_DB".Array_S7[1].rGross_Weight)
      { S7_Templates := "SrcType := Int" } NE_Contact(in1 := 0, in2 := "CylinderSetup_DB".Array_S7[4].iCylinderType)
      { S7_Templates := "SrcType := Real" } NE_Contact(in1 := 10.0, in2 := "CylinderSetup_DB".Array_S7[4].rGross_Weight)
      { S7_Templates := "SrcType := Int" } NE_Contact(in1 := 0, in2 := "CylinderSetup_DB".Array_S7[5].iCylinderType)
      { S7_Templates := "SrcType := Real" } NE_Contact(in1 := 10.0, in2 := "CylinderSetup_DB".Array_S7[5].rGross_Weight)
      { S7_Templates := "SrcType := Int" } NE_Contact(in1 := 0, in2 := "CylinderSetup_DB".Array_S7[6].iCylinderType)
      { S7_Templates := "SrcType := Real" } NE_Contact(in1 := 10.0, in2 := "CylinderSetup_DB".Array_S7[6].rGross_Weight)
      S_Coil( "Production_report_DB".Line_2_fill_done )
   END_RUNG
   RUNG wire#w1
      Contact( "Production_report_DB".Line_2_fill_done )
      { S7_Templates := "time_type := Time" } "IEC_Timer_0_DB_6".TON(pt := T#30s, et =>)
      P_Trig( "hmi_dummy_array".p_trig[3] )
      wire#w2
      R_Coil( "Production_report_DB".Line_2_fill_done )
   END_RUNG
   RUNG wire#w2
      MOVE_BLK_VARIANT(SRC := "CylinderSetup_DB".Array_S10, COUNT := 6, SRC_INDEX := 1, DEST_INDEX := 0, Ret_Val => #TEMP_5, DEST => "Production_report_DB".Production_line_2_Data)
   END_RUNG
   // the same network as SCL:
   IF true AND (0 <> "CylinderSetup_DB".Array_S7[1].iCylinderType) AND (10.0 <> "CylinderSetup_DB".Array_S7[1].rGross_Weight) AND (0 <> "CylinderSetup_DB".Array_S7[2].iCylinderType) AND (10.0 <> "CylinderSetup_DB".Array_S7[2].rGross_Weight) AND (0 <> "CylinderSetup_DB".Array_S7[3].iCylinderType) AND (10.0 <> "CylinderSetup_DB".Array_S7[1].rGross_Weight) AND (0 <> "CylinderSetup_DB".Array_S7[4].iCylinderType) AND (10.0 <> "CylinderSetup_DB".Array_S7[4].rGross_Weight) AND (0 <> "CylinderSetup_DB".Array_S7[5].iCylinderType) AND (10.0 <> "CylinderSetup_DB".Array_S7[5].rGross_Weight) AND (0 <> "CylinderSetup_DB".Array_S7[6].iCylinderType) AND (10.0 <> "CylinderSetup_DB".Array_S7[6].rGross_Weight) THEN
       "Production_report_DB".Line_2_fill_done := TRUE;
   END_IF;
   "IEC_Timer_0_DB_6".TON(IN := true AND "Production_report_DB".Line_2_fill_done, PT := T#30s);
   #_w1 := "IEC_Timer_0_DB_6".Q AND NOT "hmi_dummy_array".p_trig[3];   // rising edge
   "hmi_dummy_array".p_trig[3] := "IEC_Timer_0_DB_6".Q;
   IF #_w1 THEN
       "Production_report_DB".Line_2_fill_done := FALSE;
       #TEMP_5 := MOVE_BLK_VARIANT(SRC := "CylinderSetup_DB".Array_S10,
                               COUNT := 6,
                               SRC_INDEX := 1,
                               DEST_INDEX := 0,
                               DEST => "Production_report_DB".Production_line_2_Data);
   END_IF;
END_REGION

REGION Network 31
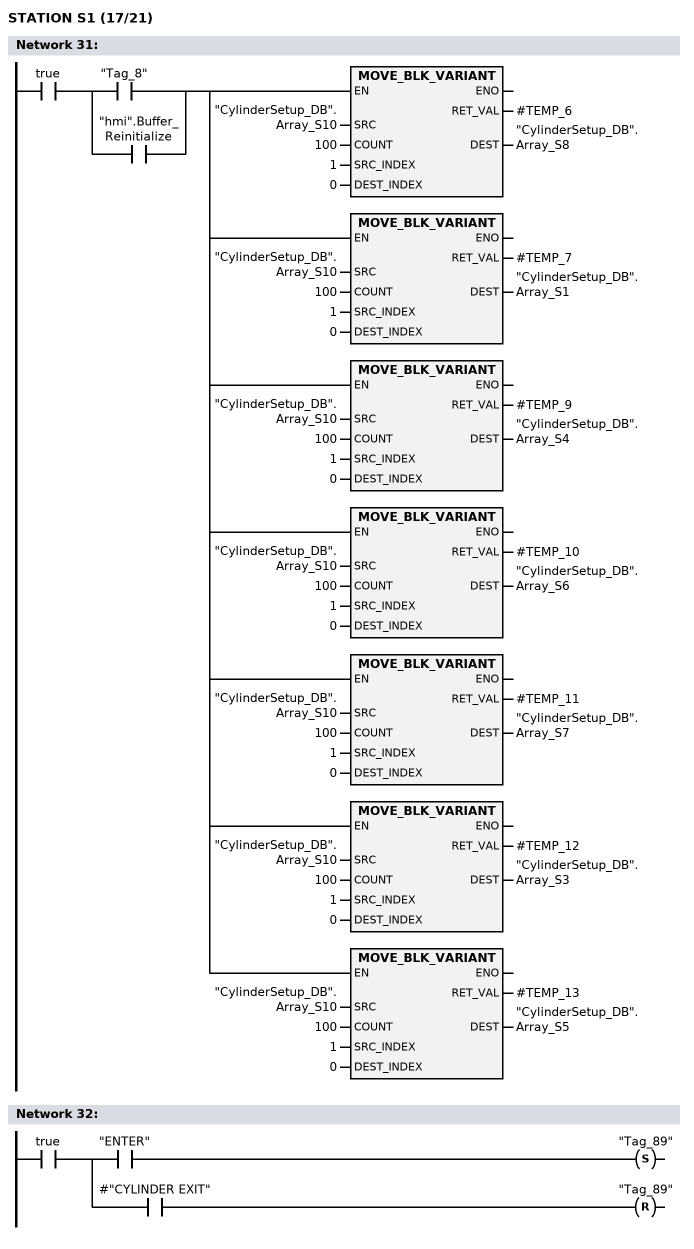
   RUNG wire#powerrail
      Contact( true )
      wire#w1
      Contact( "Tag_8" )
      wire#w2
      MOVE_BLK_VARIANT(SRC := "CylinderSetup_DB".Array_S10, COUNT := 100, SRC_INDEX := 1, DEST_INDEX := 0, Ret_Val => #TEMP_6, DEST => "CylinderSetup_DB".Array_S8)
   END_RUNG
   RUNG wire#w1
      Contact( "hmi".Buffer_Reinitialize )
   END_RUNG wire#w2
   RUNG wire#w2
      MOVE_BLK_VARIANT(SRC := "CylinderSetup_DB".Array_S10, COUNT := 100, SRC_INDEX := 1, DEST_INDEX := 0, Ret_Val => #TEMP_7, DEST => "CylinderSetup_DB".Array_S1)
   END_RUNG
   RUNG wire#w2
      MOVE_BLK_VARIANT(SRC := "CylinderSetup_DB".Array_S10, COUNT := 100, SRC_INDEX := 1, DEST_INDEX := 0, Ret_Val => #TEMP_9, DEST => "CylinderSetup_DB".Array_S4)
   END_RUNG
   RUNG wire#w2
      MOVE_BLK_VARIANT(SRC := "CylinderSetup_DB".Array_S10, COUNT := 100, SRC_INDEX := 1, DEST_INDEX := 0, Ret_Val => #TEMP_10, DEST => "CylinderSetup_DB".Array_S6)
   END_RUNG
   RUNG wire#w2
      MOVE_BLK_VARIANT(SRC := "CylinderSetup_DB".Array_S10, COUNT := 100, SRC_INDEX := 1, DEST_INDEX := 0, Ret_Val => #TEMP_11, DEST => "CylinderSetup_DB".Array_S7)
   END_RUNG
   RUNG wire#w2
      MOVE_BLK_VARIANT(SRC := "CylinderSetup_DB".Array_S10, COUNT := 100, SRC_INDEX := 1, DEST_INDEX := 0, Ret_Val => #TEMP_12, DEST => "CylinderSetup_DB".Array_S3)
   END_RUNG
   RUNG wire#w2
      MOVE_BLK_VARIANT(SRC := "CylinderSetup_DB".Array_S10, COUNT := 100, SRC_INDEX := 1, DEST_INDEX := 0, Ret_Val => #TEMP_13, DEST => "CylinderSetup_DB".Array_S5)
   END_RUNG
   // the same network as SCL:
   #_w1 := true AND ("Tag_8" OR "hmi".Buffer_Reinitialize);
   IF #_w1 THEN
       #TEMP_6 := MOVE_BLK_VARIANT(SRC := "CylinderSetup_DB".Array_S10,
                               COUNT := 100,
                               SRC_INDEX := 1,
                               DEST_INDEX := 0,
                               DEST => "CylinderSetup_DB".Array_S8);
       #TEMP_7 := MOVE_BLK_VARIANT(SRC := "CylinderSetup_DB".Array_S10,
                               COUNT := 100,
                               SRC_INDEX := 1,
                               DEST_INDEX := 0,
                               DEST => "CylinderSetup_DB".Array_S1);
       #TEMP_9 := MOVE_BLK_VARIANT(SRC := "CylinderSetup_DB".Array_S10,
                               COUNT := 100,
                               SRC_INDEX := 1,
                               DEST_INDEX := 0,
                               DEST => "CylinderSetup_DB".Array_S4);
       #TEMP_10 := MOVE_BLK_VARIANT(SRC := "CylinderSetup_DB".Array_S10,
                               COUNT := 100,
                               SRC_INDEX := 1,
                               DEST_INDEX := 0,
                               DEST => "CylinderSetup_DB".Array_S6);
       #TEMP_11 := MOVE_BLK_VARIANT(SRC := "CylinderSetup_DB".Array_S10,
                               COUNT := 100,
                               SRC_INDEX := 1,
                               DEST_INDEX := 0,
                               DEST => "CylinderSetup_DB".Array_S7);
       #TEMP_12 := MOVE_BLK_VARIANT(SRC := "CylinderSetup_DB".Array_S10,
                               COUNT := 100,
                               SRC_INDEX := 1,
                               DEST_INDEX := 0,
                               DEST => "CylinderSetup_DB".Array_S3);
       #TEMP_13 := MOVE_BLK_VARIANT(SRC := "CylinderSetup_DB".Array_S10,
                               COUNT := 100,
                               SRC_INDEX := 1,
                               DEST_INDEX := 0,
                               DEST => "CylinderSetup_DB".Array_S5);
   END_IF;
END_REGION

REGION Network 32
   RUNG wire#powerrail
      Contact( true )
      wire#w1
      Contact( "ENTER" )
      S_Coil( "Tag_89" )
   END_RUNG
   RUNG wire#w1
      Contact( #"CYLINDER EXIT" )
      R_Coil( "Tag_89" )
   END_RUNG
   // the same network as SCL:
   IF true AND "ENTER" THEN "Tag_89" := TRUE; END_IF;
   IF true AND #"CYLINDER EXIT" THEN "Tag_89" := FALSE; END_IF;
END_REGION

REGION Network 33
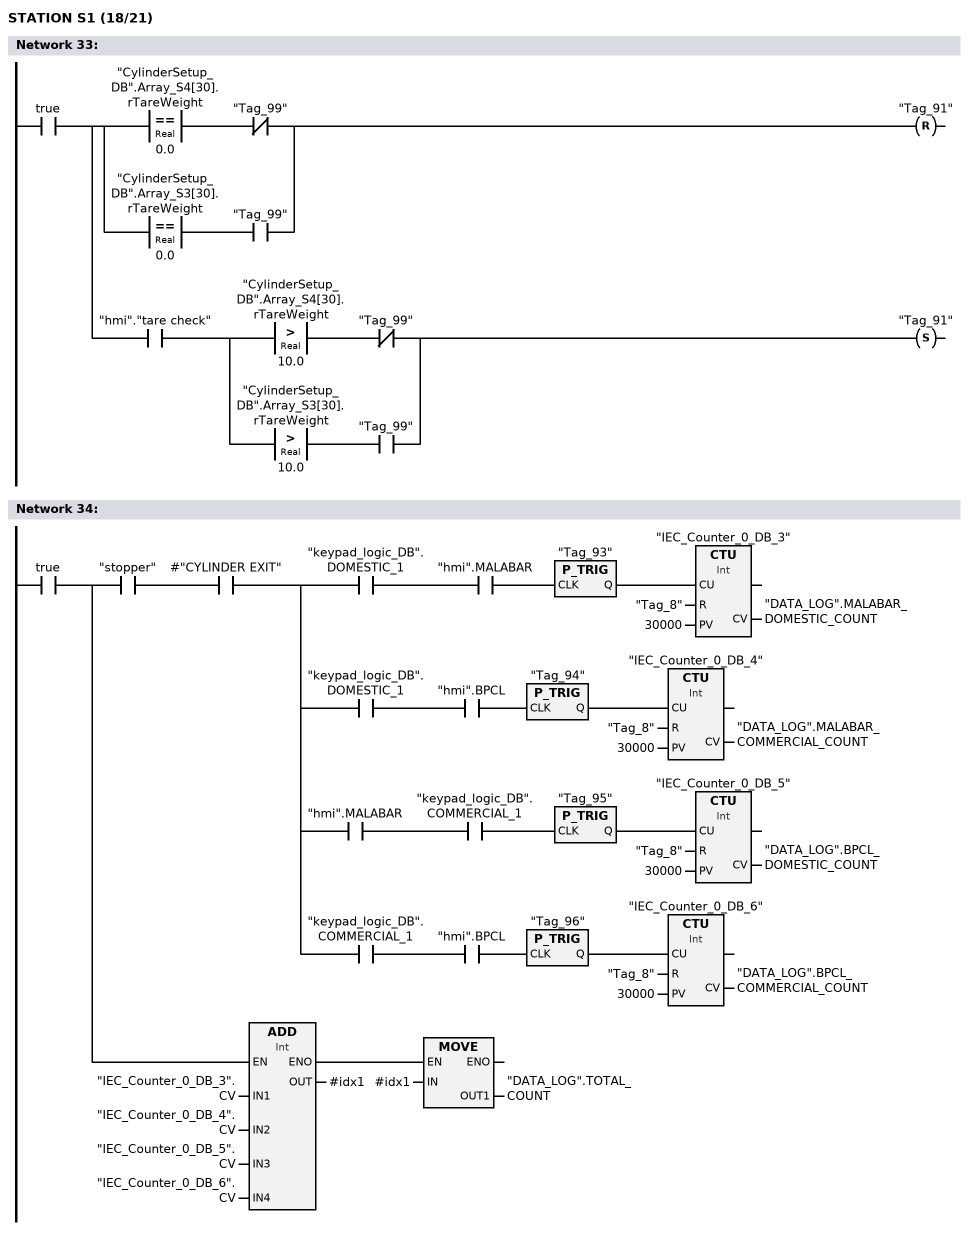
   RUNG wire#powerrail
      Contact( true )
      wire#w1
      { S7_Templates := "SrcType := Real" } EQ_Contact(in1 := "CylinderSetup_DB".Array_S4[30].rTareWeight, in2 := 0.0)
      I_Contact( "Tag_99" )
      wire#w2
      R_Coil( "Tag_91" )
   END_RUNG
   RUNG wire#w1
      { S7_Templates := "SrcType := Real" } EQ_Contact(in1 := "CylinderSetup_DB".Array_S3[30].rTareWeight, in2 := 0.0)
      Contact( "Tag_99" )
   END_RUNG wire#w2
   RUNG wire#w1
      Contact( "hmi"."tare check" )
      wire#w3
      { S7_Templates := "SrcType := Real" } GT_Contact(in1 := "CylinderSetup_DB".Array_S4[30].rTareWeight, in2 := 10.0)
      I_Contact( "Tag_99" )
      wire#w4
      S_Coil( "Tag_91" )
   END_RUNG
   RUNG wire#w3
      { S7_Templates := "SrcType := Real" } GT_Contact(in1 := "CylinderSetup_DB".Array_S3[30].rTareWeight, in2 := 10.0)
      Contact( "Tag_99" )
   END_RUNG wire#w4
   // the same network as SCL:
   IF true AND ((("CylinderSetup_DB".Array_S4[30].rTareWeight = 0.0) AND NOT "Tag_99") OR (("CylinderSetup_DB".Array_S3[30].rTareWeight = 0.0) AND "Tag_99")) THEN
       "Tag_91" := FALSE;
   END_IF;
   IF true AND "hmi"."tare check" AND ((("CylinderSetup_DB".Array_S4[30].rTareWeight > 10.0) AND NOT "Tag_99") OR (("CylinderSetup_DB".Array_S3[30].rTareWeight > 10.0) AND "Tag_99")) THEN
       "Tag_91" := TRUE;
   END_IF;
END_REGION

REGION Network 34
   RUNG wire#powerrail
      Contact( true )
      wire#w1
      Contact( "stopper" )
      Contact( #"CYLINDER EXIT" )
      wire#w2
      Contact( "keypad_logic_DB".DOMESTIC_1 )
      Contact( "hmi".MALABAR )
      P_Trig( "Tag_93" )
      { S7_Templates := "value_type := Int" } "IEC_Counter_0_DB_3".CTU(r := "Tag_8", pv := 30000, cv => "DATA_LOG".MALABAR_DOMESTIC_COUNT)
   END_RUNG
   RUNG wire#w2
      Contact( "keypad_logic_DB".DOMESTIC_1 )
      Contact( "hmi".BPCL )
      P_Trig( "Tag_94" )
      { S7_Templates := "value_type := Int" } "IEC_Counter_0_DB_4".CTU(r := "Tag_8", pv := 30000, cv => "DATA_LOG".MALABAR_COMMERCIAL_COUNT)
   END_RUNG
   RUNG wire#w2
      Contact( "hmi".MALABAR )
      Contact( "keypad_logic_DB".COMMERCIAL_1 )
      P_Trig( "Tag_95" )
      { S7_Templates := "value_type := Int" } "IEC_Counter_0_DB_5".CTU(r := "Tag_8", pv := 30000, cv => "DATA_LOG".BPCL_DOMESTIC_COUNT)
   END_RUNG
   RUNG wire#w2
      Contact( "keypad_logic_DB".COMMERCIAL_1 )
      Contact( "hmi".BPCL )
      P_Trig( "Tag_96" )
      { S7_Templates := "value_type := Int" } "IEC_Counter_0_DB_6".CTU(r := "Tag_8", pv := 30000, cv => "DATA_LOG".BPCL_COMMERCIAL_COUNT)
   END_RUNG
   RUNG wire#w1
      { S7_Templates := "SrcType := Int" } Add(in1 := "IEC_Counter_0_DB_3".CV, in2 := "IEC_Counter_0_DB_4".CV, in3 := "IEC_Counter_0_DB_5".CV, in4 := "IEC_Counter_0_DB_6".CV, out => #idx1)
      Move(in := #idx1, out1 => "DATA_LOG".TOTAL_COUNT)
   END_RUNG
   // the same network as SCL:
   #_w1 := true AND "stopper" AND #"CYLINDER EXIT";
   #_w2 := #_w1 AND "keypad_logic_DB".DOMESTIC_1 AND "hmi".MALABAR;
   #_w3 := #_w2 AND NOT "Tag_93";   // rising edge
   "Tag_93" := #_w2;
   "IEC_Counter_0_DB_3".CTU(CU := #_w3, R := "Tag_8", PV := 30000, CV => "DATA_LOG".MALABAR_DOMESTIC_COUNT);
   #_w4 := #_w1 AND "keypad_logic_DB".DOMESTIC_1 AND "hmi".BPCL;
   #_w5 := #_w4 AND NOT "Tag_94";   // rising edge
   "Tag_94" := #_w4;
   "IEC_Counter_0_DB_4".CTU(CU := #_w5, R := "Tag_8", PV := 30000, CV => "DATA_LOG".MALABAR_COMMERCIAL_COUNT);
   #_w6 := #_w1 AND "hmi".MALABAR AND "keypad_logic_DB".COMMERCIAL_1;
   #_w7 := #_w6 AND NOT "Tag_95";   // rising edge
   "Tag_95" := #_w6;
   "IEC_Counter_0_DB_5".CTU(CU := #_w7, R := "Tag_8", PV := 30000, CV => "DATA_LOG".BPCL_DOMESTIC_COUNT);
   #_w8 := #_w1 AND "keypad_logic_DB".COMMERCIAL_1 AND "hmi".BPCL;
   #_w9 := #_w8 AND NOT "Tag_96";   // rising edge
   "Tag_96" := #_w8;
   "IEC_Counter_0_DB_6".CTU(CU := #_w9, R := "Tag_8", PV := 30000, CV => "DATA_LOG".BPCL_COMMERCIAL_COUNT);
   IF true THEN
       #idx1 := "IEC_Counter_0_DB_3".CV + "IEC_Counter_0_DB_4".CV + "IEC_Counter_0_DB_5".CV + "IEC_Counter_0_DB_6".CV;
       "DATA_LOG".TOTAL_COUNT := #idx1;
   END_IF;
END_REGION

REGION Network 35: L1 TOTAL NET WT
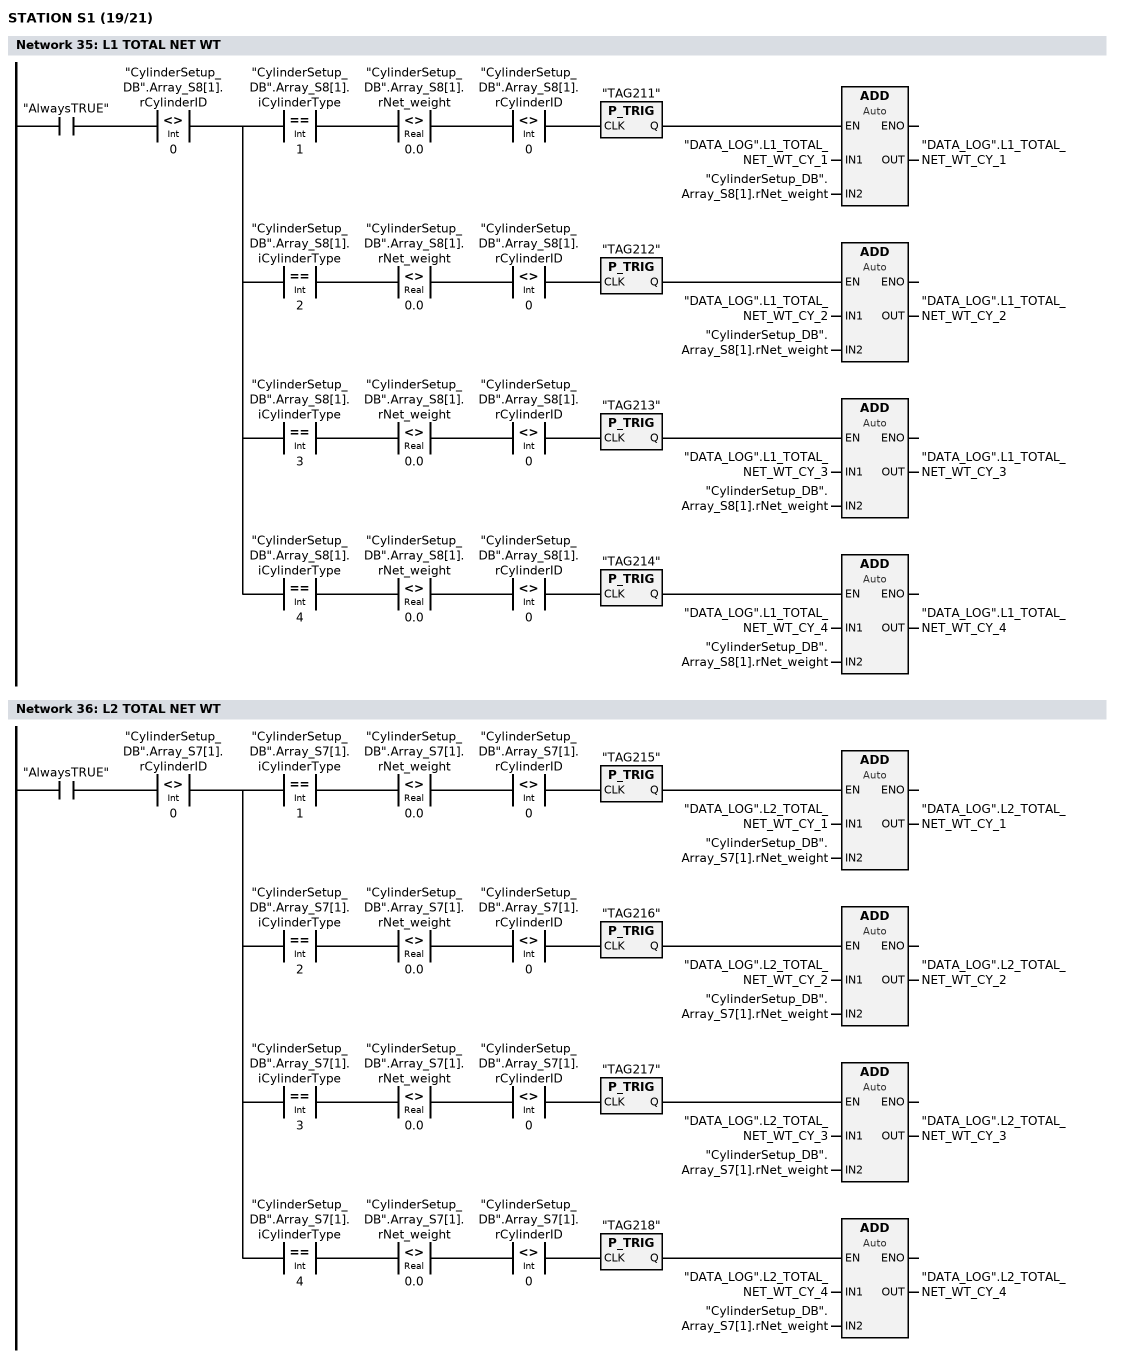
   RUNG wire#powerrail
      Contact( "AlwaysTRUE" )
      { S7_Templates := "SrcType := Int" } NE_Contact(in1 := "CylinderSetup_DB".Array_S8[1].rCylinderID, in2 := 0)
      wire#w1
      { S7_Templates := "SrcType := Int" } EQ_Contact(in1 := "CylinderSetup_DB".Array_S8[1].iCylinderType, in2 := 1)
      { S7_Templates := "SrcType := Real" } NE_Contact(in1 := "CylinderSetup_DB".Array_S8[1].rNet_weight, in2 := 0.0)
      { S7_Templates := "SrcType := Int" } NE_Contact(in1 := "CylinderSetup_DB".Array_S8[1].rCylinderID, in2 := 0)
      P_Trig( "TAG211" )
      Add(in1 := "DATA_LOG".L1_TOTAL_NET_WT_CY_1, in2 := "CylinderSetup_DB".Array_S8[1].rNet_weight, out => "DATA_LOG".L1_TOTAL_NET_WT_CY_1)
   END_RUNG
   RUNG wire#w1
      { S7_Templates := "SrcType := Int" } EQ_Contact(in1 := "CylinderSetup_DB".Array_S8[1].iCylinderType, in2 := 2)
      { S7_Templates := "SrcType := Real" } NE_Contact(in1 := "CylinderSetup_DB".Array_S8[1].rNet_weight, in2 := 0.0)
      { S7_Templates := "SrcType := Int" } NE_Contact(in1 := "CylinderSetup_DB".Array_S8[1].rCylinderID, in2 := 0)
      P_Trig( "TAG212" )
      Add(in1 := "DATA_LOG".L1_TOTAL_NET_WT_CY_2, in2 := "CylinderSetup_DB".Array_S8[1].rNet_weight, out => "DATA_LOG".L1_TOTAL_NET_WT_CY_2)
   END_RUNG
   RUNG wire#w1
      { S7_Templates := "SrcType := Int" } EQ_Contact(in1 := "CylinderSetup_DB".Array_S8[1].iCylinderType, in2 := 3)
      { S7_Templates := "SrcType := Real" } NE_Contact(in1 := "CylinderSetup_DB".Array_S8[1].rNet_weight, in2 := 0.0)
      { S7_Templates := "SrcType := Int" } NE_Contact(in1 := "CylinderSetup_DB".Array_S8[1].rCylinderID, in2 := 0)
      P_Trig( "TAG213" )
      Add(in1 := "DATA_LOG".L1_TOTAL_NET_WT_CY_3, in2 := "CylinderSetup_DB".Array_S8[1].rNet_weight, out => "DATA_LOG".L1_TOTAL_NET_WT_CY_3)
   END_RUNG
   RUNG wire#w1
      { S7_Templates := "SrcType := Int" } EQ_Contact(in1 := "CylinderSetup_DB".Array_S8[1].iCylinderType, in2 := 4)
      { S7_Templates := "SrcType := Real" } NE_Contact(in1 := "CylinderSetup_DB".Array_S8[1].rNet_weight, in2 := 0.0)
      { S7_Templates := "SrcType := Int" } NE_Contact(in1 := "CylinderSetup_DB".Array_S8[1].rCylinderID, in2 := 0)
      P_Trig( "TAG214" )
      Add(in1 := "DATA_LOG".L1_TOTAL_NET_WT_CY_4, in2 := "CylinderSetup_DB".Array_S8[1].rNet_weight, out => "DATA_LOG".L1_TOTAL_NET_WT_CY_4)
   END_RUNG
   // the same network as SCL:
   #_w1 := "AlwaysTRUE" AND ("CylinderSetup_DB".Array_S8[1].rCylinderID <> 0);
   #_w2 := #_w1 AND ("CylinderSetup_DB".Array_S8[1].iCylinderType = 1) AND ("CylinderSetup_DB".Array_S8[1].rNet_weight <> 0.0) AND ("CylinderSetup_DB".Array_S8[1].rCylinderID <> 0);
   #_w3 := #_w2 AND NOT "TAG211";   // rising edge
   "TAG211" := #_w2;
   IF #_w3 THEN
       "DATA_LOG".L1_TOTAL_NET_WT_CY_1 := "DATA_LOG".L1_TOTAL_NET_WT_CY_1 + "CylinderSetup_DB".Array_S8[1].rNet_weight;
   END_IF;
   #_w4 := #_w1 AND ("CylinderSetup_DB".Array_S8[1].iCylinderType = 2) AND ("CylinderSetup_DB".Array_S8[1].rNet_weight <> 0.0) AND ("CylinderSetup_DB".Array_S8[1].rCylinderID <> 0);
   #_w5 := #_w4 AND NOT "TAG212";   // rising edge
   "TAG212" := #_w4;
   IF #_w5 THEN
       "DATA_LOG".L1_TOTAL_NET_WT_CY_2 := "DATA_LOG".L1_TOTAL_NET_WT_CY_2 + "CylinderSetup_DB".Array_S8[1].rNet_weight;
   END_IF;
   #_w6 := #_w1 AND ("CylinderSetup_DB".Array_S8[1].iCylinderType = 3) AND ("CylinderSetup_DB".Array_S8[1].rNet_weight <> 0.0) AND ("CylinderSetup_DB".Array_S8[1].rCylinderID <> 0);
   #_w7 := #_w6 AND NOT "TAG213";   // rising edge
   "TAG213" := #_w6;
   IF #_w7 THEN
       "DATA_LOG".L1_TOTAL_NET_WT_CY_3 := "DATA_LOG".L1_TOTAL_NET_WT_CY_3 + "CylinderSetup_DB".Array_S8[1].rNet_weight;
   END_IF;
   #_w8 := #_w1 AND ("CylinderSetup_DB".Array_S8[1].iCylinderType = 4) AND ("CylinderSetup_DB".Array_S8[1].rNet_weight <> 0.0) AND ("CylinderSetup_DB".Array_S8[1].rCylinderID <> 0);
   #_w9 := #_w8 AND NOT "TAG214";   // rising edge
   "TAG214" := #_w8;
   IF #_w9 THEN
       "DATA_LOG".L1_TOTAL_NET_WT_CY_4 := "DATA_LOG".L1_TOTAL_NET_WT_CY_4 + "CylinderSetup_DB".Array_S8[1].rNet_weight;
   END_IF;
END_REGION

REGION Network 36: L2 TOTAL NET WT
   RUNG wire#powerrail
      Contact( "AlwaysTRUE" )
      { S7_Templates := "SrcType := Int" } NE_Contact(in1 := "CylinderSetup_DB".Array_S7[1].rCylinderID, in2 := 0)
      wire#w1
      { S7_Templates := "SrcType := Int" } EQ_Contact(in1 := "CylinderSetup_DB".Array_S7[1].iCylinderType, in2 := 1)
      { S7_Templates := "SrcType := Real" } NE_Contact(in1 := "CylinderSetup_DB".Array_S7[1].rNet_weight, in2 := 0.0)
      { S7_Templates := "SrcType := Int" } NE_Contact(in1 := "CylinderSetup_DB".Array_S7[1].rCylinderID, in2 := 0)
      P_Trig( "TAG215" )
      Add(in1 := "DATA_LOG".L2_TOTAL_NET_WT_CY_1, in2 := "CylinderSetup_DB".Array_S7[1].rNet_weight, out => "DATA_LOG".L2_TOTAL_NET_WT_CY_1)
   END_RUNG
   RUNG wire#w1
      { S7_Templates := "SrcType := Int" } EQ_Contact(in1 := "CylinderSetup_DB".Array_S7[1].iCylinderType, in2 := 2)
      { S7_Templates := "SrcType := Real" } NE_Contact(in1 := "CylinderSetup_DB".Array_S7[1].rNet_weight, in2 := 0.0)
      { S7_Templates := "SrcType := Int" } NE_Contact(in1 := "CylinderSetup_DB".Array_S7[1].rCylinderID, in2 := 0)
      P_Trig( "TAG216" )
      Add(in1 := "DATA_LOG".L2_TOTAL_NET_WT_CY_2, in2 := "CylinderSetup_DB".Array_S7[1].rNet_weight, out => "DATA_LOG".L2_TOTAL_NET_WT_CY_2)
   END_RUNG
   RUNG wire#w1
      { S7_Templates := "SrcType := Int" } EQ_Contact(in1 := "CylinderSetup_DB".Array_S7[1].iCylinderType, in2 := 3)
      { S7_Templates := "SrcType := Real" } NE_Contact(in1 := "CylinderSetup_DB".Array_S7[1].rNet_weight, in2 := 0.0)
      { S7_Templates := "SrcType := Int" } NE_Contact(in1 := "CylinderSetup_DB".Array_S7[1].rCylinderID, in2 := 0)
      P_Trig( "TAG217" )
      Add(in1 := "DATA_LOG".L2_TOTAL_NET_WT_CY_3, in2 := "CylinderSetup_DB".Array_S7[1].rNet_weight, out => "DATA_LOG".L2_TOTAL_NET_WT_CY_3)
   END_RUNG
   RUNG wire#w1
      { S7_Templates := "SrcType := Int" } EQ_Contact(in1 := "CylinderSetup_DB".Array_S7[1].iCylinderType, in2 := 4)
      { S7_Templates := "SrcType := Real" } NE_Contact(in1 := "CylinderSetup_DB".Array_S7[1].rNet_weight, in2 := 0.0)
      { S7_Templates := "SrcType := Int" } NE_Contact(in1 := "CylinderSetup_DB".Array_S7[1].rCylinderID, in2 := 0)
      P_Trig( "TAG218" )
      Add(in1 := "DATA_LOG".L2_TOTAL_NET_WT_CY_4, in2 := "CylinderSetup_DB".Array_S7[1].rNet_weight, out => "DATA_LOG".L2_TOTAL_NET_WT_CY_4)
   END_RUNG
   // the same network as SCL:
   #_w1 := "AlwaysTRUE" AND ("CylinderSetup_DB".Array_S7[1].rCylinderID <> 0);
   #_w2 := #_w1 AND ("CylinderSetup_DB".Array_S7[1].iCylinderType = 1) AND ("CylinderSetup_DB".Array_S7[1].rNet_weight <> 0.0) AND ("CylinderSetup_DB".Array_S7[1].rCylinderID <> 0);
   #_w3 := #_w2 AND NOT "TAG215";   // rising edge
   "TAG215" := #_w2;
   IF #_w3 THEN
       "DATA_LOG".L2_TOTAL_NET_WT_CY_1 := "DATA_LOG".L2_TOTAL_NET_WT_CY_1 + "CylinderSetup_DB".Array_S7[1].rNet_weight;
   END_IF;
   #_w4 := #_w1 AND ("CylinderSetup_DB".Array_S7[1].iCylinderType = 2) AND ("CylinderSetup_DB".Array_S7[1].rNet_weight <> 0.0) AND ("CylinderSetup_DB".Array_S7[1].rCylinderID <> 0);
   #_w5 := #_w4 AND NOT "TAG216";   // rising edge
   "TAG216" := #_w4;
   IF #_w5 THEN
       "DATA_LOG".L2_TOTAL_NET_WT_CY_2 := "DATA_LOG".L2_TOTAL_NET_WT_CY_2 + "CylinderSetup_DB".Array_S7[1].rNet_weight;
   END_IF;
   #_w6 := #_w1 AND ("CylinderSetup_DB".Array_S7[1].iCylinderType = 3) AND ("CylinderSetup_DB".Array_S7[1].rNet_weight <> 0.0) AND ("CylinderSetup_DB".Array_S7[1].rCylinderID <> 0);
   #_w7 := #_w6 AND NOT "TAG217";   // rising edge
   "TAG217" := #_w6;
   IF #_w7 THEN
       "DATA_LOG".L2_TOTAL_NET_WT_CY_3 := "DATA_LOG".L2_TOTAL_NET_WT_CY_3 + "CylinderSetup_DB".Array_S7[1].rNet_weight;
   END_IF;
   #_w8 := #_w1 AND ("CylinderSetup_DB".Array_S7[1].iCylinderType = 4) AND ("CylinderSetup_DB".Array_S7[1].rNet_weight <> 0.0) AND ("CylinderSetup_DB".Array_S7[1].rCylinderID <> 0);
   #_w9 := #_w8 AND NOT "TAG218";   // rising edge
   "TAG218" := #_w8;
   IF #_w9 THEN
       "DATA_LOG".L2_TOTAL_NET_WT_CY_4 := "DATA_LOG".L2_TOTAL_NET_WT_CY_4 + "CylinderSetup_DB".Array_S7[1].rNet_weight;
   END_IF;
END_REGION

REGION Network 37
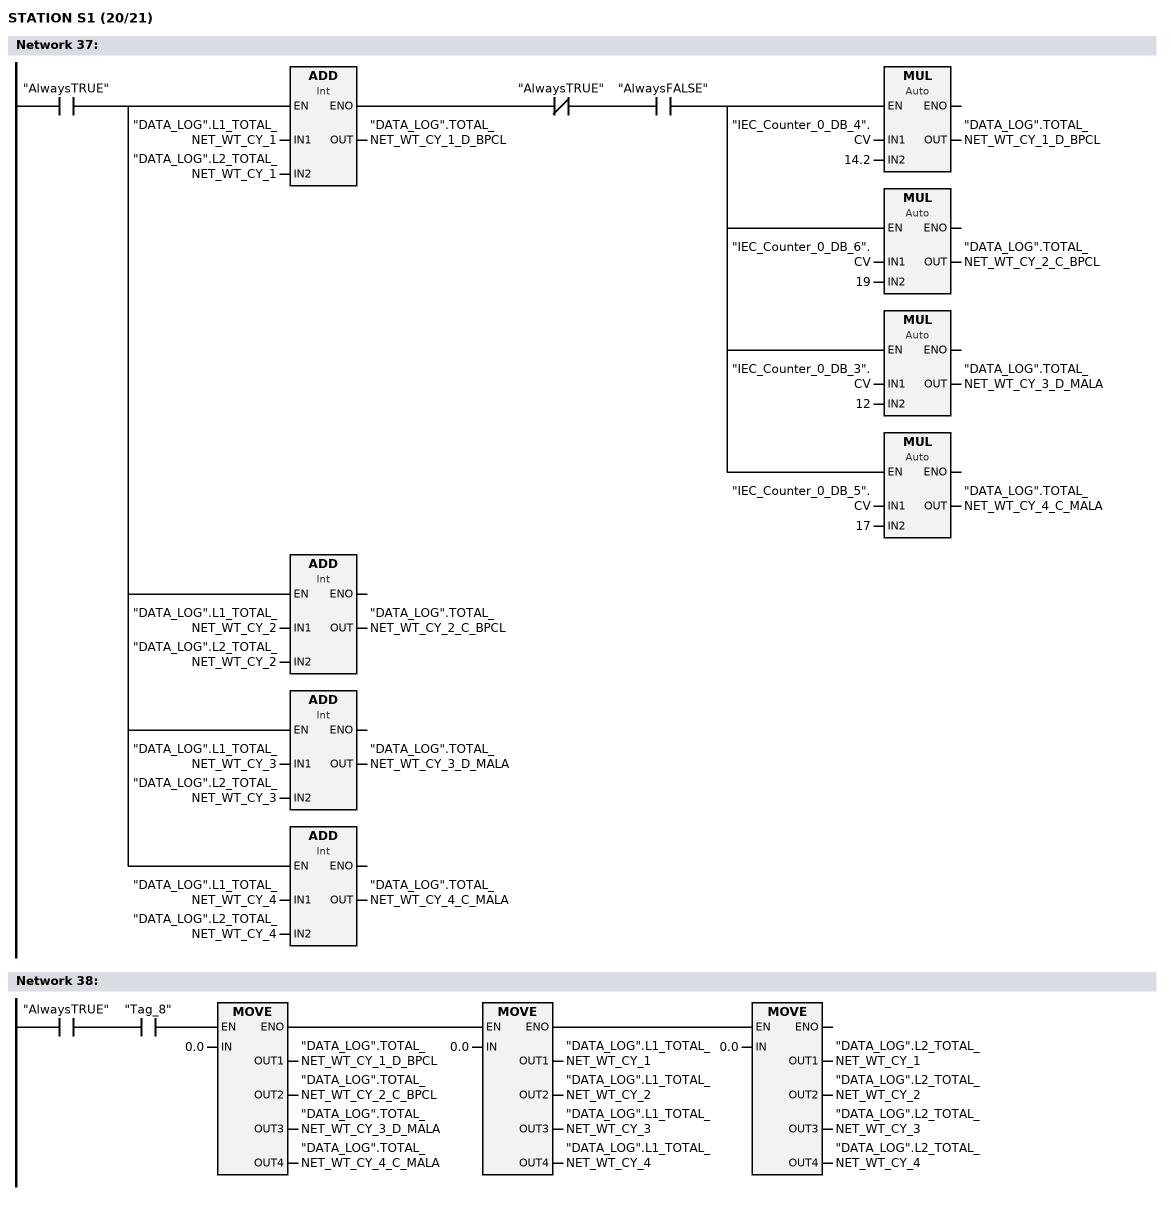
   RUNG wire#powerrail
      Contact( "AlwaysTRUE" )
      wire#w1
      { S7_Templates := "SrcType := Int" } Add(in1 := "DATA_LOG".L1_TOTAL_NET_WT_CY_1, in2 := "DATA_LOG".L2_TOTAL_NET_WT_CY_1, out => "DATA_LOG".TOTAL_NET_WT_CY_1_D_BPCL)
      I_Contact( "AlwaysTRUE" )
      Contact( "AlwaysFALSE" )
      wire#w2
      Mul(in1 := "IEC_Counter_0_DB_4".CV, in2 := 14.2, out => "DATA_LOG".TOTAL_NET_WT_CY_1_D_BPCL)
   END_RUNG
   RUNG wire#w2
      Mul(in1 := "IEC_Counter_0_DB_6".CV, in2 := 19, out => "DATA_LOG".TOTAL_NET_WT_CY_2_C_BPCL)
   END_RUNG
   RUNG wire#w2
      Mul(in1 := "IEC_Counter_0_DB_3".CV, in2 := 12, out => "DATA_LOG".TOTAL_NET_WT_CY_3_D_MALA)
   END_RUNG
   RUNG wire#w2
      Mul(in1 := "IEC_Counter_0_DB_5".CV, in2 := 17, out => "DATA_LOG".TOTAL_NET_WT_CY_4_C_MALA)
   END_RUNG
   RUNG wire#w1
      { S7_Templates := "SrcType := Int" } Add(in1 := "DATA_LOG".L1_TOTAL_NET_WT_CY_2, in2 := "DATA_LOG".L2_TOTAL_NET_WT_CY_2, out => "DATA_LOG".TOTAL_NET_WT_CY_2_C_BPCL)
   END_RUNG
   RUNG wire#w1
      { S7_Templates := "SrcType := Int" } Add(in1 := "DATA_LOG".L1_TOTAL_NET_WT_CY_3, in2 := "DATA_LOG".L2_TOTAL_NET_WT_CY_3, out => "DATA_LOG".TOTAL_NET_WT_CY_3_D_MALA)
   END_RUNG
   RUNG wire#w1
      { S7_Templates := "SrcType := Int" } Add(in1 := "DATA_LOG".L1_TOTAL_NET_WT_CY_4, in2 := "DATA_LOG".L2_TOTAL_NET_WT_CY_4, out => "DATA_LOG".TOTAL_NET_WT_CY_4_C_MALA)
   END_RUNG
   // the same network as SCL:
   IF "AlwaysTRUE" THEN
       "DATA_LOG".TOTAL_NET_WT_CY_1_D_BPCL := "DATA_LOG".L1_TOTAL_NET_WT_CY_1 + "DATA_LOG".L2_TOTAL_NET_WT_CY_1;
   END_IF;
   IF "AlwaysTRUE" AND NOT "AlwaysTRUE" AND "AlwaysFALSE" THEN
       "DATA_LOG".TOTAL_NET_WT_CY_1_D_BPCL := "IEC_Counter_0_DB_4".CV * 14.2;
       "DATA_LOG".TOTAL_NET_WT_CY_2_C_BPCL := "IEC_Counter_0_DB_6".CV * 19;
       "DATA_LOG".TOTAL_NET_WT_CY_3_D_MALA := "IEC_Counter_0_DB_3".CV * 12;
       "DATA_LOG".TOTAL_NET_WT_CY_4_C_MALA := "IEC_Counter_0_DB_5".CV * 17;
   END_IF;
   IF "AlwaysTRUE" THEN
       "DATA_LOG".TOTAL_NET_WT_CY_2_C_BPCL := "DATA_LOG".L1_TOTAL_NET_WT_CY_2 + "DATA_LOG".L2_TOTAL_NET_WT_CY_2;
       "DATA_LOG".TOTAL_NET_WT_CY_3_D_MALA := "DATA_LOG".L1_TOTAL_NET_WT_CY_3 + "DATA_LOG".L2_TOTAL_NET_WT_CY_3;
       "DATA_LOG".TOTAL_NET_WT_CY_4_C_MALA := "DATA_LOG".L1_TOTAL_NET_WT_CY_4 + "DATA_LOG".L2_TOTAL_NET_WT_CY_4;
   END_IF;
END_REGION

REGION Network 38
   RUNG wire#powerrail
      Contact( "AlwaysTRUE" )
      Contact( "Tag_8" )
      Move(in := 0.0, out1 => "DATA_LOG".TOTAL_NET_WT_CY_1_D_BPCL, out2 => "DATA_LOG".TOTAL_NET_WT_CY_2_C_BPCL, out3 => "DATA_LOG".TOTAL_NET_WT_CY_3_D_MALA, out4 => "DATA_LOG".TOTAL_NET_WT_CY_4_C_MALA)
      Move(in := 0.0, out1 => "DATA_LOG".L1_TOTAL_NET_WT_CY_1, out2 => "DATA_LOG".L1_TOTAL_NET_WT_CY_2, out3 => "DATA_LOG".L1_TOTAL_NET_WT_CY_3, out4 => "DATA_LOG".L1_TOTAL_NET_WT_CY_4)
      Move(in := 0.0, out1 => "DATA_LOG".L2_TOTAL_NET_WT_CY_1, out2 => "DATA_LOG".L2_TOTAL_NET_WT_CY_2, out3 => "DATA_LOG".L2_TOTAL_NET_WT_CY_3, out4 => "DATA_LOG".L2_TOTAL_NET_WT_CY_4)
   END_RUNG
   // the same network as SCL:
   IF "AlwaysTRUE" AND "Tag_8" THEN
       "DATA_LOG".TOTAL_NET_WT_CY_1_D_BPCL := 0.0;
       "DATA_LOG".TOTAL_NET_WT_CY_2_C_BPCL := 0.0;
       "DATA_LOG".TOTAL_NET_WT_CY_3_D_MALA := 0.0;
       "DATA_LOG".TOTAL_NET_WT_CY_4_C_MALA := 0.0;
       "DATA_LOG".L1_TOTAL_NET_WT_CY_1 := 0.0;
       "DATA_LOG".L1_TOTAL_NET_WT_CY_2 := 0.0;
       "DATA_LOG".L1_TOTAL_NET_WT_CY_3 := 0.0;
       "DATA_LOG".L1_TOTAL_NET_WT_CY_4 := 0.0;
       "DATA_LOG".L2_TOTAL_NET_WT_CY_1 := 0.0;
       "DATA_LOG".L2_TOTAL_NET_WT_CY_2 := 0.0;
       "DATA_LOG".L2_TOTAL_NET_WT_CY_3 := 0.0;
       "DATA_LOG".L2_TOTAL_NET_WT_CY_4 := 0.0;
   END_IF;
END_REGION

REGION Network 39: filled CYL data to check scale data
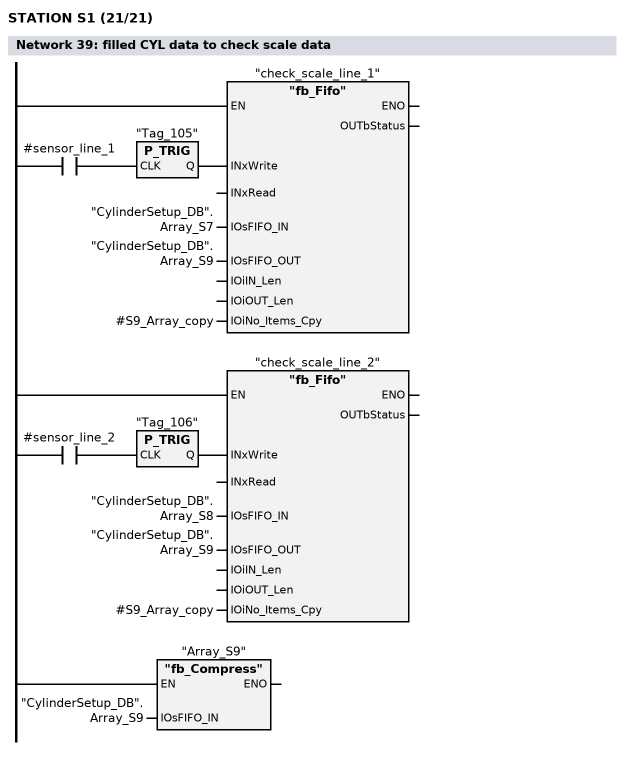
   RUNG wire#powerrail
      "check_scale_line_1"(INxWrite := wire#w1, INxRead :=, IOsFIFO_IN := "CylinderSetup_DB".Array_S7, IOsFIFO_OUT := "CylinderSetup_DB".Array_S9, IOiIN_Len :=, IOiOUT_Len :=, IOiNo_Items_Cpy := #S9_Array_copy, OUTbStatus =>)
   END_RUNG
   RUNG wire#powerrail
      Contact( #sensor_line_1 )
      P_Trig( "Tag_105" )
   END_RUNG wire#w1
   RUNG wire#powerrail
      "check_scale_line_2"(INxWrite := wire#w2, INxRead :=, IOsFIFO_IN := "CylinderSetup_DB".Array_S8, IOsFIFO_OUT := "CylinderSetup_DB".Array_S9, IOiIN_Len :=, IOiOUT_Len :=, IOiNo_Items_Cpy := #S9_Array_copy, OUTbStatus =>)
   END_RUNG
   RUNG wire#powerrail
      Contact( #sensor_line_2 )
      P_Trig( "Tag_106" )
   END_RUNG wire#w2
   RUNG wire#powerrail
      "Array_S9"(IOsFIFO_IN := "CylinderSetup_DB".Array_S9)
   END_RUNG
   // the same network as SCL:
   #_w1 := #sensor_line_1 AND NOT "Tag_105";   // rising edge
   "Tag_105" := #sensor_line_1;
   "check_scale_line_1"(INxWrite := #_w1,   // "fb_Fifo"
                        IOsFIFO_IN := "CylinderSetup_DB".Array_S7,
                        IOsFIFO_OUT := "CylinderSetup_DB".Array_S9,
                        IOiNo_Items_Cpy := #S9_Array_copy);
   #_w2 := #sensor_line_2 AND NOT "Tag_106";   // rising edge
   "Tag_106" := #sensor_line_2;
   "check_scale_line_2"(INxWrite := #_w2,   // "fb_Fifo"
                        IOsFIFO_IN := "CylinderSetup_DB".Array_S8,
                        IOsFIFO_OUT := "CylinderSetup_DB".Array_S9,
                        IOiNo_Items_Cpy := #S9_Array_copy);
   "Array_S9"(IOsFIFO_IN := "CylinderSetup_DB".Array_S9);   // "fb_Compress"
END_REGION
END_FUNCTION
